KUKA KRL program: MyProgram_023().src

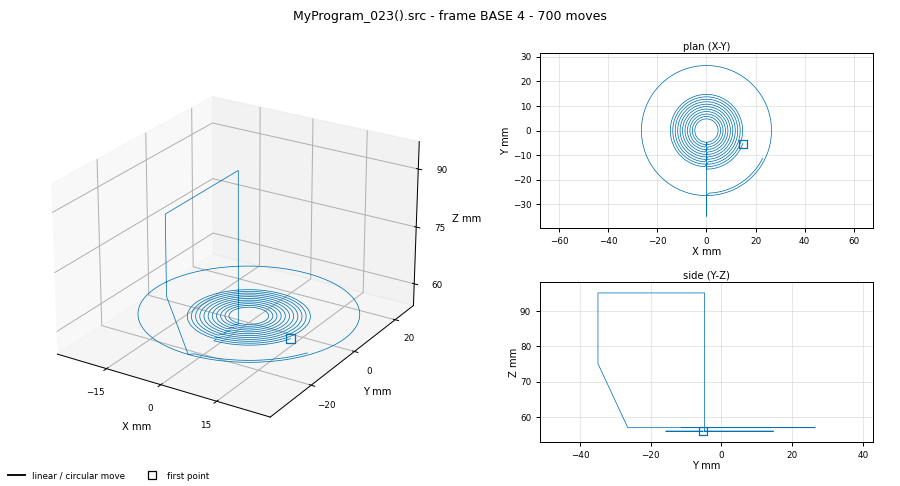
[picture p0: tool path of MyProgram_023().src in frame BASE 4, 700 of 700 moves have a stored position in this frame; points joined in program order, loops and branches not executed]
&ACCESS RVP
&REL 1
&PARAM TEMPLATE = C:\KRC\Roboter\Template\vorgabe
&PARAM EDITMASK = *
DEF MyProgram_023()
; ---- Setting reference (Base) ----
$BASE = BASE_DATA[4]

; --------------------------
; ---- Setting tool (TCP) ----
$TOOL = TOOL_DATA[3]
; --------------------------

$VEL.CP = VEL_APROX_PRINT
Startdeposition()
$VEL.CP = VEL_PRINT
LIN {X 14.8048,Y -5.3302,Z 56,A -29.3112,B 24.8121,C -3.1607,E1 25.1484,E2 -248.3313} C_DIS
LIN {X 13.9602,Y -7.2597,Z 56,A -35.481,B 24.8134,C -3.1503,E1 25.1412,E2 -242.1703} C_DIS
LIN {X 13.4677,Y -8.1371,Z 56,A -39.3253,B 24.8148,C -3.1386,E1 25.1358,E2 -238.3181} C_DIS
LIN {X 12.8219,Y -9.1209,Z 56,A -44.2575,B 24.8167,C -3.122,E1 25.128,E2 -233.371} C_DIS
LIN {X 12.0786,Y -10.0846,Z 56,A -48.5761,B 24.818,C -3.1116,E1 25.1204,E2 -229.0476} C_DIS
LIN {X 11.0622,Y -11.1901,Z 56,A -53.5865,B 24.8191,C -3.1018,E1 25.1107,E2 -224.0359} C_DIS
LIN {X 10.1799,Y -11.9958,Z 56,A -57.8584,B 24.8202,C -3.0927,E1 25.1018,E2 -219.7593} C_DIS
LIN {X 9.2719,Y -12.7131,Z 56,A -62.3619,B 24.8214,C -3.0819,E1 25.0918,E2 -215.2466} C_DIS
LIN {X 8.1629,Y -13.4521,Z 56,A -67.2273,B 24.8225,C -3.0728,E1 25.0803,E2 -210.3752} C_DIS
LIN {X 7.0535,Y -14.0655,Z 56,A -71.7054,B 24.8233,C -3.0661,E1 25.0693,E2 -205.8939} C_DIS
LIN {X 5.5713,Y -14.7154,Z 56,A -78.5194,B 24.8249,C -3.0521,E1 25.0516,E2 -199.062} C_DIS
LIN {X 4.0025,Y -15.2173,Z 56,A -84.3756,B 24.8255,C -3.0465,E1 25.0359,E2 -193.2024} C_DIS
LIN {X 1.9688,Y -15.6113,Z 56,A -91.411,B 24.8258,C -3.044,E1 25.0165,E2 -186.168} C_DIS
LIN {X 0.1829,Y -15.7341,Z 56,A -98.106,B 24.8262,C -3.0407,E1 24.9978,E2 -179.4672} C_DIS
LIN {X 0.1829,Y -15.7341,Z 56,A -98.106,B 24.8262,C -3.0407,E1 24.9978,E2 -179.4672} C_DIS
Enddeposition()
LIN {X 0.0548,Y -14.7363,Z 56,A -95.9481,B 24.8226,C -3.0715,E1 25.004,E2 -181.6985} C_DIS
Startdeposition()
$VEL.CP = VEL_PRINT
LIN {X 1.2094,Y -14.6873,Z 56,A -90.7717,B 24.822,C -3.0772,E1 25.0185,E2 -186.886} C_DIS
LIN {X 3.1948,Y -14.3867,Z 56,A -83.0175,B 24.8213,C -3.083,E1 25.0398,E2 -194.6453} C_DIS
LIN {X 4.7095,Y -13.964,Z 56,A -77.5601,B 24.821,C -3.0859,E1 25.0543,E2 -200.0999} C_DIS
LIN {X 5.781,Y -13.5555,Z 56,A -72.1308,B 24.8195,C -3.0983,E1 25.0684,E2 -205.5461} C_DIS
LIN {X 7.833,Y -12.4829,Z 56,A -64.8508,B 24.8191,C -3.1022,E1 25.0861,E2 -212.8139} C_DIS
LIN {X 8.8701,Y -11.7687,Z 56,A -58.779,B 24.817,C -3.12,E1 25.1,E2 -218.907} C_DIS
LIN {X 9.9895,Y -10.8348,Z 56,A -53.7158,B 24.816,C -3.1283,E1 25.1106,E2 -223.9698} C_DIS
LIN {X 10.8598,Y -9.9602,Z 56,A -49.2201,B 24.8149,C -3.1375,E1 25.1193,E2 -228.4681} C_DIS
LIN {X 11.6373,Y -9.042,Z 56,A -44.418,B 24.8134,C -3.1504,E1 25.1279,E2 -233.2784} C_DIS
LIN {X 12.467,Y -7.8585,Z 56,A -37.7373,B 24.8106,C -3.1737,E1 25.1382,E2 -239.9813} C_DIS
LIN {X 13.1856,Y -6.5817,Z 56,A -32.3096,B 24.8089,C -3.1879,E1 25.1452,E2 -245.4139} C_DIS
LIN {X 13.8526,Y -5.0285,Z 56,A -26.548,B 24.8073,C -3.201,E1 25.1512,E2 -251.1747} C_DIS
LIN {X 14.1872,Y -3.9875,Z 56,A -22.1497,B 24.8056,C -3.2151,E1 25.1547,E2 -255.5813} C_DIS
LIN {X 14.4328,Y -2.9781,Z 56,A -18.2812,B 24.8042,C -3.2262,E1 25.1571,E2 -259.4536} C_DIS
LIN {X 14.6165,Y -1.8806,Z 56,A -13.1649,B 24.8018,C -3.246,E1 25.1591,E2 -264.5866} C_DIS
LIN {X 14.7344,Y -0.2827,Z 56,A -7.0232,B 24.7995,C -3.2646,E1 25.1598,E2 -270.7361} C_DIS
LIN {X 14.6312,Y 1.7639,Z 56,A 0.269,B 24.7972,C -3.2837,E1 25.1582,E2 -278.0303} C_DIS
LIN {X 14.3689,Y 3.2719,Z 56,A 6.2117,B 24.7949,C -3.3016,E1 25.155,E2 -283.9807} C_DIS
LIN {X 13.964,Y 4.709,Z 56,A 12.9283,B 24.7919,C -3.3256,E1 25.1494,E2 -290.716} C_DIS
LIN {X 13.275,Y 6.3989,Z 56,A 18.77,B 24.7907,C -3.3355,E1 25.1428,E2 -296.5494} C_DIS
LIN {X 12.5995,Y 7.6442,Z 56,A 25.1855,B 24.788,C -3.3565,E1 25.1338,E2 -302.9817} C_DIS
LIN {X 11.6707,Y 8.9959,Z 56,A 29.6616,B 24.7878,C -3.3581,E1 25.1266,E2 -307.4397} C_DIS
LIN {X 10.7914,Y 10.0362,Z 56,A 37.2967,B 24.7842,C -3.3862,E1 25.1125,E2 -315.1075} C_DIS
LIN {X 9.6504,Y 11.138,Z 56,A 42.6202,B 24.7834,C -3.3923,E1 25.1014,E2 -320.4241} C_DIS
LIN {X 8.5044,Y 12.0354,Z 56,A 47.752,B 24.7827,C -3.3985,E1 25.09,E2 -325.552} C_DIS
LIN {X 7.3595,Y 12.7674,Z 56,A 53.871,B 24.781,C -3.4113,E1 25.0753,E2 -331.6826} C_DIS
LIN {X 5.1068,Y 13.8238,Z 56,A 64.3115,B 24.7791,C -3.4257,E1 25.0484,E2 -342.133} C_DIS
LIN {X 3.3707,Y 14.3465,Z 56,A 69.8758,B 24.7796,C -3.4218,E1 25.0335,E2 -347.6792} C_DIS
LIN {X 2.2012,Y 14.5718,Z 56,A 74.8904,B 24.7792,C -3.4253,E1 25.0196,E2 -352.6969} C_DIS
LIN {X 0.5459,Y 14.7267,Z 56,A 80.5918,B 24.7796,C -3.4218,E1 25.0038,E2 -358.3873} C_DIS
LIN {X -0.7491,Y 14.7179,Z 56,A 86.5134,B 24.7793,C -3.4244,E1 24.9873,E2 -364.3159} C_DIS
LIN {X -1.8751,Y 14.6172,Z 56,A 90.6939,B 24.7797,C -3.421,E1 24.9757,E2 -368.4912} C_DIS
LIN {X -3.2885,Y 14.3633,Z 56,A 95.6264,B 24.7807,C -3.414,E1 24.9622,E2 -373.4124} C_DIS
LIN {X -4.3601,Y 14.0772,Z 56,A 100.1365,B 24.7811,C -3.4102,E1 24.9501,E2 -377.9208} C_DIS
LIN {X -5.4825,Y 13.6792,Z 56,A 104.5629,B 24.782,C -3.4036,E1 24.9385,E2 -382.3406} C_DIS
LIN {X -6.4904,Y 13.2307,Z 56,A 109.4506,B 24.7826,C -3.3992,E1 24.9262,E2 -387.2301} C_DIS
LIN {X -7.726,Y 12.5494,Z 56,A 115.2787,B 24.7836,C -3.3908,E1 24.9122,E2 -393.0555} C_DIS
LIN {X -9.1952,Y 11.5166,Z 56,A 121.4568,B 24.7857,C -3.3745,E1 24.8983,E2 -399.2167} C_DIS
LIN {X -10.1448,Y 10.6894,Z 56,A 127.0188,B 24.7869,C -3.3654,E1 24.8868,E2 -404.7791} C_DIS
LIN {X -11.2667,Y 9.4995,Z 56,A 133.2509,B 24.7889,C -3.3495,E1 24.8752,E2 -411.0011} C_DIS
LIN {X -12.1246,Y 8.377,Z 56,A 138.6054,B 24.7908,C -3.3348,E1 24.8664,E2 -416.3463} C_DIS
LIN {X -12.8562,Y 7.2042,Z 56,A 144.3048,B 24.7925,C -3.3206,E1 24.8583,E2 -422.0411} C_DIS
LIN {X -13.4172,Y 6.096,Z 56,A 148.769,B 24.7944,C -3.306,E1 24.853,E2 -426.4944} C_DIS
LIN {X -13.8066,Y 5.153,Z 56,A 152.7105,B 24.7959,C -3.2942,E1 24.849,E2 -430.4297} C_DIS
LIN {X -14.0831,Y 4.3412,Z 56,A 156.2898,B 24.7971,C -3.2846,E1 24.8459,E2 -434.0065} C_DIS
LIN {X -14.4046,Y 3.1126,Z 56,A 160.9881,B 24.799,C -3.269,E1 24.8429,E2 -438.6951} C_DIS
LIN {X -14.6238,Y 1.8249,Z 56,A 166.5143,B 24.8008,C -3.2541,E1 24.8406,E2 -444.2183} C_DIS
LIN {X -14.7274,Y 0.4637,Z 56,A 171.4099,B 24.8029,C -3.2369,E1 24.8398,E2 -449.1022} C_DIS
LIN {X -14.7165,Y -0.7763,Z 56,A 176.4141,B 24.8047,C -3.2223,E1 24.8402,E2 -454.1014} C_DIS
LIN {X -14.6103,Y -1.9279,Z 56,A -178.8358,B 24.8063,C -3.209,E1 24.8417,E2 -458.848} C_DIS
LIN {X -14.3442,Y -3.3805,Z 56,A -173.1358,B 24.8084,C -3.1917,E1 24.8449,E2 -464.5403} C_DIS
LIN {X -14.0463,Y -4.4582,Z 56,A -168.0512,B 24.8098,C -3.1805,E1 24.849,E2 -469.6274} C_DIS
LIN {X -13.3291,Y -6.2865,Z 56,A -161.3284,B 24.8125,C -3.1574,E1 24.8563,E2 -476.332} C_DIS
LIN {X -12.9229,Y -7.0841,Z 56,A -156.6672,B 24.8133,C -3.1509,E1 24.8625,E2 -481.0023} C_DIS
LIN {X -11.7295,Y -8.9216,Z 56,A -149.7736,B 24.8162,C -3.1261,E1 24.8733,E2 -487.8708} C_DIS
LIN {X -11.1715,Y -9.6111,Z 56,A -144.1744,B 24.8165,C -3.1243,E1 24.8835,E2 -493.491} C_DIS
LIN {X -9.3084,Y -11.4252,Z 56,A -135.6271,B 24.8193,C -3.1,E1 24.901,E2 -502.0148} C_DIS
LIN {X -8.4511,Y -12.0728,Z 56,A -130.3651,B 24.8197,C -3.0967,E1 24.913,E2 -507.2873} C_DIS
LIN {X -6.7508,Y -13.0998,Z 56,A -123.6353,B 24.8213,C -3.0828,E1 24.9293,E2 -514.0036} C_DIS
LIN {X -5.8273,Y -13.5357,Z 56,A -119.2256,B 24.8216,C -3.0803,E1 24.9405,E2 -518.4179} C_DIS
LIN {X -4.5384,Y -14.0208,Z 56,A -113.6765,B 24.822,C -3.0768,E1 24.9551,E2 -523.9693} C_DIS
LIN {X -2.9742,Y -14.4336,Z 56,A -107.9788,B 24.8227,C -3.071,E1 24.9706,E2 -529.661} C_DIS
LIN {X -1.9619,Y -14.6057,Z 56,A -103.8651,B 24.8227,C -3.0706,E1 24.982,E2 -533.7773} C_DIS
LIN {X -0.703,Y -14.7188,Z 56,A -99.2648,B 24.8229,C -3.069,E1 24.9948,E2 -538.3758} C_DIS
LIN {X -0.703,Y -14.7188,Z 56,A -99.2648,B 24.8229,C -3.069,E1 24.9948,E2 -538.3758} C_DIS
Enddeposition()
LIN {X 0.0882,Y -13.7373,Z 56,A -99.2033,B 24.8225,C -3.0726,E1 24.995,E2 -538.4457} C_DIS
Startdeposition()
$VEL.CP = VEL_PRINT
LIN {X -2.2045,Y -13.5607,Z 56,A -108.546,B 24.8223,C -3.0749,E1 24.9691,E2 -529.1025} C_DIS
LIN {X -3.6611,Y -13.242,Z 56,A -113.9205,B 24.8215,C -3.0814,E1 24.9545,E2 -523.7359} C_DIS
LIN {X -4.8429,Y -12.8549,Z 56,A -118,B 24.8206,C -3.0895,E1 24.9438,E2 -519.6682} C_DIS
LIN {X -5.7969,Y -12.4563,Z 56,A -124.0655,B 24.8207,C -3.0881,E1 24.9282,E2 -513.5848} C_DIS
LIN {X -6.9738,Y -11.8372,Z 56,A -129.4609,B 24.8198,C -3.0959,E1 24.9151,E2 -508.1924} C_DIS
LIN {X -8.2177,Y -11.0106,Z 56,A -135.281,B 24.8185,C -3.107,E1 24.9018,E2 -502.3788} C_DIS
LIN {X -9.1001,Y -10.293,Z 56,A -140.145,B 24.8175,C -3.1154,E1 24.8915,E2 -497.5162} C_DIS
LIN {X -9.9975,Y -9.4238,Z 56,A -145.2366,B 24.8162,C -3.1264,E1 24.8815,E2 -492.4291} C_DIS
LIN {X -10.7189,Y -8.5947,Z 56,A -150.0677,B 24.8151,C -3.1361,E1 24.8728,E2 -487.5991} C_DIS
LIN {X -11.4994,Y -7.5177,Z 56,A -154.969,B 24.8133,C -3.1508,E1 24.865,E2 -482.709} C_DIS
LIN {X -12.258,Y -6.2049,Z 56,A -162.1921,B 24.8115,C -3.1657,E1 24.8553,E2 -475.4836} C_DIS
LIN {X -12.8192,Y -4.9422,Z 56,A -167.9265,B 24.8096,C -3.1818,E1 24.8491,E2 -469.7559} C_DIS
LIN {X -13.2224,Y -3.7266,Z 56,A -171.871,B 24.8075,C -3.1994,E1 24.8458,E2 -465.8309} C_DIS
LIN {X -13.4775,Y -2.6674,Z 56,A -178.6467,B 24.8062,C -3.2099,E1 24.8418,E2 -459.0404} C_DIS
LIN {X -13.6777,Y -1.296,Z 56,A 175.7485,B 24.804,C -3.2278,E1 24.8401,E2 -453.4449} C_DIS
LIN {X -13.7274,Y 0.565,Z 56,A 168.6555,B 24.801,C -3.2527,E1 24.8401,E2 -446.3689} C_DIS
LIN {X -13.6144,Y 1.8474,Z 56,A 163.0023,B 24.799,C -3.269,E1 24.8419,E2 -440.721} C_DIS
LIN {X -13.4072,Y 3.0004,Z 56,A 158.4536,B 24.7971,C -3.2844,E1 24.8444,E2 -436.1826} C_DIS
LIN {X -13.1292,Y 4.048,Z 56,A 153.6733,B 24.7954,C -3.2978,E1 24.8481,E2 -431.4067} C_DIS
LIN {X -12.5255,Y 5.6457,Z 56,A 146.1859,B 24.7928,C -3.3183,E1 24.856,E2 -423.9267} C_DIS
LIN {X -11.7299,Y 7.1534,Z 56,A 139.5054,B 24.7903,C -3.3389,E1 24.8651,E2 -417.2604} C_DIS
LIN {X -11.0348,Y 8.1853,Z 56,A 132.9569,B 24.7888,C -3.3503,E1 24.8758,E2 -410.7074} C_DIS
LIN {X -9.4035,Y 10.0169,Z 56,A 123.6703,B 24.7855,C -3.3764,E1 24.8936,E2 -401.4431} C_DIS
LIN {X -8.4735,Y 10.815,Z 56,A 118.8118,B 24.784,C -3.3877,E1 24.9041,E2 -396.5934} C_DIS
LIN {X -7.5312,Y 11.4909,Z 56,A 113.8264,B 24.7829,C -3.3966,E1 24.9156,E2 -391.6126} C_DIS
LIN {X -6.3763,Y 12.1697,Z 56,A 108.8007,B 24.7815,C -3.4075,E1 24.9278,E2 -386.5983} C_DIS
LIN {X -5.4377,Y 12.617,Z 56,A 103.8915,B 24.7809,C -3.4122,E1 24.9402,E2 -381.6883} C_DIS
LIN {X -4.2833,Y 13.0522,Z 56,A 99.2225,B 24.7799,C -3.42,E1 24.9525,E2 -377.0287} C_DIS
LIN {X -3.3313,Y 13.3291,Z 56,A 94.4774,B 24.7796,C -3.422,E1 24.9653,E2 -372.2812} C_DIS
LIN {X -2.0113,Y 13.5886,Z 56,A 89.4219,B 24.7788,C -3.4282,E1 24.9792,E2 -367.2353} C_DIS
LIN {X -0.6959,Y 13.7213,Z 56,A 83.4729,B 24.7788,C -3.4289,E1 24.9957,E2 -361.2853} C_DIS
LIN {X 0.2866,Y 13.7361,Z 56,A 79.6032,B 24.7785,C -3.4305,E1 25.0065,E2 -357.4199} C_DIS
LIN {X 1.5068,Y 13.6561,Z 56,A 74.0874,B 24.7788,C -3.4283,E1 25.0218,E2 -351.9018} C_DIS
LIN {X 2.9208,Y 13.425,Z 56,A 68.1409,B 24.7791,C -3.4261,E1 25.0381,E2 -345.957} C_DIS
LIN {X 4.6649,Y 12.9228,Z 56,A 59.697,B 24.7804,C -3.4159,E1 25.0606,E2 -337.5044} C_DIS
LIN {X 6.2714,Y 12.2241,Z 56,A 53.4336,B 24.7808,C -3.4132,E1 25.0764,E2 -331.2508} C_DIS
LIN {X 7.31,Y 11.633,Z 56,A 48.2066,B 24.7819,C -3.4046,E1 25.0889,E2 -326.0197} C_DIS
LIN {X 8.7427,Y 10.5986,Z 56,A 42.1869,B 24.7824,C -3.4003,E1 25.1023,E2 -320.0114} C_DIS
LIN {X 9.9736,Y 9.4495,Z 56,A 32.2437,B 24.7866,C -3.3674,E1 25.1221,E2 -310.0319} C_DIS
LIN {X 11.3157,Y 7.7921,Z 56,A 24.0158,B 24.7888,C -3.3506,E1 25.1356,E2 -301.8038} C_DIS
LIN {X 12.4931,Y 5.7173,Z 56,A 15.6873,B 24.7907,C -3.3356,E1 25.1464,E2 -293.4836} C_DIS
LIN {X 12.9049,Y 4.7075,Z 56,A 11.2831,B 24.7921,C -3.3239,E1 25.1509,E2 -289.076} C_DIS
LIN {X 13.2704,Y 3.5574,Z 56,A 6.0217,B 24.7942,C -3.3075,E1 25.1551,E2 -283.8057} C_DIS
LIN {X 13.5032,Y 2.535,Z 56,A 1.2414,B 24.7962,C -3.2913,E1 25.1578,E2 -279.0151} C_DIS
LIN {X 13.6854,Y 1.2119,Z 56,A -3.7214,B 24.7978,C -3.2788,E1 25.1594,E2 -274.0519} C_DIS
LIN {X 13.7354,Y 0.1773,Z 56,A -7.8731,B 24.7993,C -3.2667,E1 25.1598,E2 -269.8962} C_DIS
LIN {X 13.687,Y -1.1935,Z 56,A -14.0401,B 24.8019,C -3.2455,E1 25.1588,E2 -263.7156} C_DIS
LIN {X 13.5157,Y -2.4674,Z 56,A -19.5239,B 24.804,C -3.228,E1 25.1564,E2 -258.2224} C_DIS
LIN {X 13.127,Y -4.0549,Z 56,A -25.7527,B 24.806,C -3.2115,E1 25.1519,E2 -251.9904} C_DIS
LIN {X 12.7794,Y -5.0447,Z 56,A -30.7044,B 24.8081,C -3.1942,E1 25.147,E2 -247.0253} C_DIS
LIN {X 12.2474,Y -6.2256,Z 56,A -35.9164,B 24.8098,C -3.18,E1 25.1407,E2 -241.8075} C_DIS
LIN {X 11.6127,Y -7.3418,Z 56,A -41.0181,B 24.8114,C -3.1669,E1 25.1334,E2 -236.7009} C_DIS
LIN {X 10.9215,Y -8.3359,Z 56,A -45.6641,B 24.8127,C -3.1564,E1 25.1258,E2 -232.0524} C_DIS
LIN {X 10.082,Y -9.3337,Z 56,A -51.3966,B 24.8145,C -3.1408,E1 25.1152,E2 -226.3088} C_DIS
LIN {X 9.1447,Y -10.2537,Z 56,A -57.3574,B 24.8164,C -3.125,E1 25.1031,E2 -220.335} C_DIS
LIN {X 8.074,Y -11.116,Z 56,A -62.3643,B 24.8172,C -3.1179,E1 25.092,E2 -215.3294} C_DIS
LIN {X 7.3076,Y -11.6345,Z 56,A -67.32,B 24.8189,C -3.1038,E1 25.0803,E2 -210.3564} C_DIS
LIN {X 5.4767,Y -12.5999,Z 56,A -75.3509,B 24.82,C -3.0939,E1 25.0601,E2 -202.3232} C_DIS
LIN {X 3.8332,Y -13.1933,Z 56,A -82.8593,B 24.8212,C -3.084,E1 25.0402,E2 -194.8057} C_DIS
LIN {X 2.3245,Y -13.5406,Z 56,A -88.9914,B 24.8216,C -3.0803,E1 25.0234,E2 -188.6722} C_DIS
LIN {X 1.0278,Y -13.7006,Z 56,A -94.9502,B 24.8222,C -3.075,E1 25.0068,E2 -182.7043} C_DIS
LIN {X 0.0882,Y -13.7373,Z 56,A -99.2033,B 24.8225,C -3.0726,E1 24.995,E2 -178.4457} C_DIS
Enddeposition()
LIN {X 0.0882,Y -13.7373,Z 56,A -99.2033,B 24.8225,C -3.0726,E1 24.995,E2 -178.4457} C_DIS
Startdeposition()
$VEL.CP = VEL_PRINT
LIN {X 0.846,Y -12.7129,Z 56,A -92.2496,B 24.8185,C -3.1072,E1 25.0146,E2 -185.4806} C_DIS
LIN {X 2.1074,Y -12.5656,Z 56,A -85.9473,B 24.8177,C -3.114,E1 25.032,E2 -191.7932} C_DIS
LIN {X 3.68,Y -12.1981,Z 56,A -79.2495,B 24.8172,C -3.1184,E1 25.0501,E2 -198.491} C_DIS
LIN {X 4.7745,Y -11.8127,Z 56,A -73.2317,B 24.8158,C -3.1298,E1 25.0658,E2 -204.5228} C_DIS
LIN {X 6.5926,Y -10.903,Z 56,A -65.1697,B 24.8148,C -3.1386,E1 25.0856,E2 -212.5827} C_DIS
LIN {X 7.6738,Y -10.171,Z 56,A -58.5287,B 24.8128,C -3.1551,E1 25.1007,E2 -219.2397} C_DIS
LIN {X 8.7439,Y -9.2671,Z 56,A -51.5317,B 24.8106,C -3.174,E1 25.1151,E2 -226.2531} C_DIS
LIN {X 10.2047,Y -7.6288,Z 56,A -42.9898,B 24.8086,C -3.1898,E1 25.1303,E2 -234.7934} C_DIS
LIN {X 10.9664,Y -6.4864,Z 56,A -36.3429,B 24.8062,C -3.2101,E1 25.1402,E2 -241.4548} C_DIS
LIN {X 11.5007,Y -5.4837,Z 56,A -31.1854,B 24.8044,C -3.2252,E1 25.1466,E2 -246.6204} C_DIS
LIN {X 12.1365,Y -3.8775,Z 56,A -25.0553,B 24.803,C -3.2366,E1 25.1525,E2 -252.7433} C_DIS
LIN {X 12.3867,Y -2.9845,Z 56,A -20.1005,B 24.8007,C -3.255,E1 25.1561,E2 -257.7132} C_DIS
LIN {X 12.5465,Y -2.2183,Z 56,A -16.2178,B 24.799,C -3.2686,E1 25.158,E2 -261.6055} C_DIS
LIN {X 12.7239,Y -0.6578,Z 56,A -9.0136,B 24.7962,C -3.2916,E1 25.1597,E2 -268.8215} C_DIS
LIN {X 12.7133,Y 0.84,Z 56,A -2.7132,B 24.794,C -3.3092,E1 25.1591,E2 -275.1263} C_DIS
LIN {X 12.5589,Y 2.1475,Z 56,A 4.0308,B 24.791,C -3.3332,E1 25.1563,E2 -281.8875} C_DIS
LIN {X 12.0597,Y 4.1104,Z 56,A 11.3207,B 24.7892,C -3.3469,E1 25.1509,E2 -289.168} C_DIS
LIN {X 11.6949,Y 5.0558,Z 56,A 16.5606,B 24.787,C -3.3645,E1 25.1454,E2 -294.4206} C_DIS
LIN {X 11.0719,Y 6.3047,Z 56,A 23.0344,B 24.7847,C -3.3824,E1 25.1369,E2 -300.9029} C_DIS
LIN {X 10.4017,Y 7.3581,Z 56,A 28.2429,B 24.7833,C -3.3936,E1 25.1289,E2 -306.1121} C_DIS
LIN {X 9.8575,Y 8.0724,Z 56,A 33.2066,B 24.7813,C -3.4089,E1 25.1202,E2 -311.0889} C_DIS
LIN {X 8.6383,Y 9.3654,Z 56,A 40.2128,B 24.78,C -3.4191,E1 25.1064,E2 -318.0897} C_DIS
LIN {X 7.5062,Y 10.2953,Z 56,A 47.3336,B 24.7781,C -3.4339,E1 25.0907,E2 -325.2192} C_DIS
LIN {X 6.5786,Y 10.9114,Z 56,A 52.0428,B 24.7773,C -3.4396,E1 25.0796,E2 -329.927} C_DIS
LIN {X 5.4854,Y 11.4997,Z 56,A 57.6724,B 24.7764,C -3.4467,E1 25.0656,E2 -335.5582} C_DIS
LIN {X 4.2005,Y 12.0286,Z 56,A 64.408,B 24.7753,C -3.455,E1 25.048,E2 -342.2989} C_DIS
LIN {X 2.9819,Y 12.3873,Z 56,A 69.945,B 24.775,C -3.4575,E1 25.033,E2 -347.8334} C_DIS
LIN {X 1.5044,Y 12.652,Z 56,A 76.7474,B 24.7747,C -3.4595,E1 25.0143,E2 -354.6343} C_DIS
LIN {X 0.0834,Y 12.7408,Z 56,A 82.7812,B 24.775,C -3.4575,E1 24.9974,E2 -360.6618} C_DIS
LIN {X -1.2068,Y 12.6837,Z 56,A 88.7478,B 24.7752,C -3.4557,E1 24.9808,E2 -366.6264} C_DIS
LIN {X -2.5336,Y 12.4865,Z 56,A 94.8571,B 24.7758,C -3.4516,E1 24.9641,E2 -372.732} C_DIS
LIN {X -3.5731,Y 12.2296,Z 56,A 99.4798,B 24.7765,C -3.4461,E1 24.9516,E2 -377.3488} C_DIS
LIN {X -4.7424,Y 11.8255,Z 56,A 105.282,B 24.7773,C -3.4398,E1 24.9365,E2 -383.1479} C_DIS
LIN {X -5.5626,Y 11.4627,Z 56,A 110.2068,B 24.7778,C -3.436,E1 24.9241,E2 -388.0764} C_DIS
LIN {X -7.3339,Y 10.4187,Z 56,A 118.1935,B 24.7804,C -3.4161,E1 24.9053,E2 -396.041} C_DIS
LIN {X -8.226,Y 9.7299,Z 56,A 123.5553,B 24.7817,C -3.4061,E1 24.8937,E2 -401.3989} C_DIS
LIN {X -9.1126,Y 8.9049,Z 56,A 128.9947,B 24.7833,C -3.3935,E1 24.8829,E2 -406.831} C_DIS
LIN {X -9.9217,Y 7.9936,Z 56,A 134.7244,B 24.785,C -3.3803,E1 24.8726,E2 -412.5552} C_DIS
LIN {X -10.7926,Y 6.7713,Z 56,A 141.1342,B 24.7874,C -3.3617,E1 24.8626,E2 -418.9523} C_DIS
LIN {X -11.431,Y 5.627,Z 56,A 147.1457,B 24.7895,C -3.3451,E1 24.8547,E2 -424.9561} C_DIS
LIN {X -11.8217,Y 4.7523,Z 56,A 151.5735,B 24.791,C -3.3326,E1 24.85,E2 -429.3785} C_DIS
LIN {X -12.2361,Y 3.551,Z 56,A 156.9921,B 24.7932,C -3.3151,E1 24.8453,E2 -434.786} C_DIS
LIN {X -12.5152,Y 2.3885,Z 56,A 162.5489,B 24.7953,C -3.2988,E1 24.842,E2 -440.3364} C_DIS
LIN {X -12.6745,Y 1.3008,Z 56,A 168.055,B 24.7971,C -3.2841,E1 24.8402,E2 -445.8401} C_DIS
LIN {X -12.7392,Y -0.2228,Z 56,A 174.5894,B 24.7998,C -3.2624,E1 24.8399,E2 -452.362} C_DIS
LIN {X -12.6656,Y -1.3839,Z 56,A 179.7288,B 24.8018,C -3.2462,E1 24.8411,E2 -457.4934} C_DIS
LIN {X -12.5123,Y -2.4001,Z 56,A -175.4287,B 24.8035,C -3.2326,E1 24.8434,E2 -462.3319} C_DIS
LIN {X -12.1912,Y -3.7032,Z 56,A -170.2033,B 24.8058,C -3.2138,E1 24.8472,E2 -467.5427} C_DIS
LIN {X -11.8078,Y -4.7856,Z 56,A -164.107,B 24.8074,C -3.2004,E1 24.8531,E2 -473.6413} C_DIS
LIN {X -11.2481,Y -5.984,Z 56,A -158.033,B 24.8093,C -3.1847,E1 24.8607,E2 -479.7103} C_DIS
LIN {X -10.3963,Y -7.3652,Z 56,A -150.7404,B 24.8114,C -3.1666,E1 24.8718,E2 -486.9962} C_DIS
LIN {X -9.5188,Y -8.4686,Z 56,A -143.7134,B 24.813,C -3.1539,E1 24.8845,E2 -494.0249} C_DIS
LIN {X -8.0975,Y -9.8364,Z 56,A -135.2277,B 24.8151,C -3.136,E1 24.9021,E2 -502.5018} C_DIS
LIN {X -6.9871,Y -10.6542,Z 56,A -129.0524,B 24.8163,C -3.1261,E1 24.9162,E2 -508.6743} C_DIS
LIN {X -6.1846,Y -11.1395,Z 56,A -125.0349,B 24.817,C -3.1199,E1 24.926,E2 -512.6888} C_DIS
LIN {X -5.3265,Y -11.5744,Z 56,A -120.8363,B 24.8176,C -3.1145,E1 24.9366,E2 -516.8854} C_DIS
LIN {X -4.0768,Y -12.0712,Z 56,A -114.3431,B 24.8181,C -3.1109,E1 24.9536,E2 -523.383} C_DIS
LIN {X -2.7873,Y -12.4323,Z 56,A -108.7352,B 24.8186,C -3.1061,E1 24.9687,E2 -528.9875} C_DIS
LIN {X -1.7393,Y -12.6219,Z 56,A -104.0183,B 24.8188,C -3.1045,E1 24.9818,E2 -533.7049} C_DIS
LIN {X -0.655,Y -12.7241,Z 56,A -98.9908,B 24.8188,C -3.1051,E1 24.9958,E2 -538.7358} C_DIS
LIN {X -0.655,Y -12.7241,Z 56,A -98.9908,B 24.8188,C -3.1051,E1 24.9958,E2 -538.7358} C_DIS
Enddeposition()
LIN {X 0.0689,Y -11.7371,Z 56,A -96.9233,B 24.8172,C -3.1177,E1 25.0016,E2 -540.8333} C_DIS
Startdeposition()
$VEL.CP = VEL_PRINT
LIN {X -0.9726,Y -11.7024,Z 56,A -103.1695,B 24.8178,C -3.1127,E1 24.9842,E2 -534.5737} C_DIS
LIN {X -2.0877,Y -11.556,Z 56,A -109.1817,B 24.8178,C -3.1122,E1 24.9676,E2 -528.5551} C_DIS
LIN {X -3.0518,Y -11.3394,Z 56,A -114.07,B 24.8176,C -3.1146,E1 24.9543,E2 -523.6655} C_DIS
LIN {X -4.533,Y -10.8325,Z 56,A -121.9664,B 24.8169,C -3.1206,E1 24.9337,E2 -515.7672} C_DIS
LIN {X -5.6889,Y -10.2731,Z 56,A -127.7671,B 24.8159,C -3.1295,E1 24.9193,E2 -509.9718} C_DIS
LIN {X -6.6994,Y -9.6409,Z 56,A -133.2843,B 24.8147,C -3.139,E1 24.9065,E2 -504.4593} C_DIS
LIN {X -7.3672,Y -9.1412,Z 56,A -137.3038,B 24.8139,C -3.1461,E1 24.8976,E2 -500.4421} C_DIS
LIN {X -7.9978,Y -8.5953,Z 56,A -141.4431,B 24.813,C -3.1538,E1 24.889,E2 -496.3045} C_DIS
LIN {X -8.5875,Y -8.0055,Z 56,A -145.4987,B 24.812,C -3.1622,E1 24.8811,E2 -492.2518} C_DIS
LIN {X -9.1346,Y -7.376,Z 56,A -149.6163,B 24.8109,C -3.1713,E1 24.8737,E2 -488.1368} C_DIS
LIN {X -9.7547,Y -6.5378,Z 56,A -154.9489,B 24.8095,C -3.1831,E1 24.8652,E2 -482.8066} C_DIS
LIN {X -10.2644,Y -5.7047,Z 56,A -160.3975,B 24.8081,C -3.1947,E1 24.8576,E2 -477.3572} C_DIS
LIN {X -10.9919,Y -4.1321,Z 56,A -167.9347,B 24.8051,C -3.2189,E1 24.8492,E2 -469.8364} C_DIS
LIN {X -11.5022,Y -2.3647,Z 56,A -178.9176,B 24.8021,C -3.2439,E1 24.8417,E2 -458.8496} C_DIS
LIN {X -11.7262,Y -0.6128,Z 56,A 173.2612,B 24.7988,C -3.2709,E1 24.8398,E2 -451.046} C_DIS
LIN {X -11.6918,Y 1.0956,Z 56,A 164.8812,B 24.7955,C -3.2967,E1 24.8411,E2 -442.6777} C_DIS
LIN {X -11.4868,Y 2.4409,Z 56,A 158.8117,B 24.7929,C -3.3175,E1 24.8441,E2 -436.6221} C_DIS
LIN {X -11.2026,Y 3.5215,Z 56,A 153.0503,B 24.7909,C -3.3339,E1 24.8486,E2 -430.8665} C_DIS
LIN {X -10.7955,Y 4.6202,Z 56,A 147.3153,B 24.7888,C -3.3507,E1 24.8545,E2 -425.14} C_DIS
LIN {X -10.2689,Y 5.6967,Z 56,A 142.136,B 24.7866,C -3.3679,E1 24.8611,E2 -419.9742} C_DIS
LIN {X -9.5216,Y 6.8732,Z 56,A 133.2496,B 24.7845,C -3.384,E1 24.8751,E2 -411.0824} C_DIS
LIN {X -7.9763,Y 8.6186,Z 56,A 122.0094,B 24.781,C -3.411,E1 24.8969,E2 -399.8587} C_DIS
LIN {X -6.8958,Y 9.5049,Z 56,A 115.5157,B 24.7792,C -3.4253,E1 24.9114,E2 -393.3759} C_DIS
LIN {X -5.2981,Y 10.4799,Z 56,A 107.467,B 24.7769,C -3.4429,E1 24.9309,E2 -385.3458} C_DIS
LIN {X -4.3393,Y 10.9121,Z 56,A 101.5841,B 24.7762,C -3.4482,E1 24.946,E2 -379.4621} C_DIS
LIN {X -2.8904,Y 11.3818,Z 56,A 94.6219,B 24.775,C -3.4573,E1 24.9647,E2 -372.5101} C_DIS
LIN {X -1.571,Y 11.6375,Z 56,A 87.6205,B 24.7746,C -3.4605,E1 24.9839,E2 -365.5099} C_DIS
LIN {X -0.3179,Y 11.7389,Z 56,A 81.9891,B 24.7741,C -3.4644,E1 24.9996,E2 -359.8861} C_DIS
LIN {X 0.7997,Y 11.7158,Z 56,A 76.2345,B 24.7742,C -3.4635,E1 25.0157,E2 -354.1314} C_DIS
LIN {X 2.0147,Y 11.5691,Z 56,A 70.2249,B 24.7744,C -3.4618,E1 25.0322,E2 -348.1231} C_DIS
LIN {X 3.2337,Y 11.289,Z 56,A 64.5724,B 24.7746,C -3.4602,E1 25.0475,E2 -342.4753} C_DIS
LIN {X 4.1701,Y 10.9771,Z 56,A 59.0303,B 24.7756,C -3.4526,E1 25.0621,E2 -336.9268} C_DIS
LIN {X 5.8427,Y 10.1864,Z 56,A 50.4083,B 24.7768,C -3.4435,E1 25.0835,E2 -328.3067} C_DIS
LIN {X 6.9689,Y 9.4518,Z 56,A 44.2671,B 24.7779,C -3.4352,E1 25.0976,E2 -322.1668} C_DIS
LIN {X 7.932,Y 8.6594,Z 56,A 37.6415,B 24.7798,C -3.4208,E1 25.1116,E2 -315.5329} C_DIS
LIN {X 8.7174,Y 7.8682,Z 56,A 32.1301,B 24.7813,C -3.4088,E1 25.1221,E2 -310.017} C_DIS
LIN {X 9.7238,Y 6.584,Z 56,A 24.1917,B 24.7837,C -3.3899,E1 25.1352,E2 -302.0722} C_DIS
LIN {X 10.515,Y 5.2281,Z 56,A 16.7782,B 24.7861,C -3.3714,E1 25.1451,E2 -294.6534} C_DIS
LIN {X 11.0579,Y 3.9525,Z 56,A 10.0932,B 24.7885,C -3.3529,E1 25.1519,E2 -287.9616} C_DIS
LIN {X 11.3944,Y 2.8409,Z 56,A 4.7855,B 24.7903,C -3.3386,E1 25.1559,E2 -282.6506} C_DIS
LIN {X 11.593,Y 1.8704,Z 56,A -0.1487,B 24.7922,C -3.3234,E1 25.1583,E2 -277.7091} C_DIS
LIN {X 11.7215,Y 0.706,Z 56,A -5.447,B 24.7941,C -3.3086,E1 25.1596,E2 -272.4072} C_DIS
LIN {X 11.7141,Y -0.8229,Z 56,A -13.0618,B 24.7971,C -3.2844,E1 25.1591,E2 -264.7803} C_DIS
LIN {X 11.5493,Y -2.1251,Z 56,A -19.7989,B 24.7998,C -3.2623,E1 25.1563,E2 -258.0303} C_DIS
LIN {X 11.2431,Y -3.3904,Z 56,A -25.3163,B 24.8015,C -3.2485,E1 25.1523,E2 -252.5121} C_DIS
LIN {X 10.9547,Y -4.2298,Z 56,A -30.1052,B 24.8035,C -3.2325,E1 25.1478,E2 -247.7119} C_DIS
LIN {X 10.4428,Y -5.3654,Z 56,A -34.8196,B 24.8045,C -3.224,E1 25.1422,E2 -243.0029} C_DIS
LIN {X 9.9467,Y -6.242,Z 56,A -41.6782,B 24.8077,C -3.1975,E1 25.1325,E2 -236.1166} C_DIS
LIN {X 9.1352,Y -7.3789,Z 56,A -48.1538,B 24.8096,C -3.1819,E1 25.1215,E2 -229.6348} C_DIS
LIN {X 8.2431,Y -8.3638,Z 56,A -54.2695,B 24.8112,C -3.1686,E1 25.1097,E2 -223.514} C_DIS
LIN {X 7.4207,Y -9.1011,Z 56,A -59.6999,B 24.8126,C -3.1565,E1 25.0982,E2 -218.0762} C_DIS
LIN {X 6.4532,Y -9.8111,Z 56,A -64.9778,B 24.8136,C -3.1483,E1 25.0861,E2 -212.797} C_DIS
LIN {X 5.2093,Y -10.5243,Z 56,A -72.7678,B 24.8155,C -3.1322,E1 25.067,E2 -204.9912} C_DIS
LIN {X 4.0383,Y -11.0268,Z 56,A -78.8324,B 24.8164,C -3.1246,E1 25.0512,E2 -198.922} C_DIS
LIN {X 2.6585,Y -11.4381,Z 56,A -86.2807,B 24.8175,C -3.1154,E1 25.0311,E2 -191.4637} C_DIS
LIN {X 0.9818,Y -11.7016,Z 56,A -93.8354,B 24.8177,C -3.1135,E1 25.0102,E2 -183.9103} C_DIS
LIN {X 0.0689,Y -11.7371,Z 56,A -96.9233,B 24.8172,C -3.1177,E1 25.0016,E2 -180.8333} C_DIS
Enddeposition()
LIN {X 0.0689,Y -11.7371,Z 56,A -96.9233,B 24.8172,C -3.1177,E1 25.0016,E2 -180.8333} C_DIS
Startdeposition()
$VEL.CP = VEL_PRINT
LIN {X 0.4819,Y -10.7343,Z 56,A -92.7327,B 24.8142,C -3.1434,E1 25.0135,E2 -185.0837} C_DIS
LIN {X 2.1779,Y -10.5217,Z 56,A -84.8318,B 24.8141,C -3.1445,E1 25.0353,E2 -192.9798} C_DIS
LIN {X 3.5686,Y -10.1349,Z 56,A -75.7142,B 24.8122,C -3.1599,E1 25.0596,E2 -202.1177} C_DIS
LIN {X 5.1038,Y -9.4556,Z 56,A -67.7535,B 24.8112,C -3.1687,E1 25.0796,E2 -210.0783} C_DIS
LIN {X 6.0628,Y -8.8714,Z 56,A -62.4013,B 24.8103,C -3.1763,E1 25.0922,E2 -215.4315} C_DIS
LIN {X 7.2221,Y -7.9562,Z 56,A -52.4324,B 24.8067,C -3.2056,E1 25.1135,E2 -225.4312} C_DIS
LIN {X 8.4512,Y -6.6355,Z 56,A -44.354,B 24.805,C -3.2201,E1 25.1282,E2 -233.5075} C_DIS
LIN {X 9.1708,Y -5.594,Z 56,A -39.0508,B 24.8039,C -3.2293,E1 25.1365,E2 -238.8063} C_DIS
LIN {X 9.6542,Y -4.7172,Z 56,A -31.5702,B 24.8003,C -3.2582,E1 25.1462,E2 -246.316} C_DIS
LIN {X 10.2192,Y -3.3118,Z 56,A -25.7546,B 24.7992,C -3.2675,E1 25.152,E2 -252.1213} C_DIS
LIN {X 10.4244,Y -2.6067,Z 56,A -20.1964,B 24.7963,C -3.2903,E1 25.1561,E2 -257.7014} C_DIS
LIN {X 10.6471,Y -1.4317,Z 56,A -14.4932,B 24.7944,C -3.3056,E1 25.1587,E2 -263.4075} C_DIS
LIN {X 10.7433,Y -0.1964,Z 56,A -7.2552,B 24.7913,C -3.3303,E1 25.1598,E2 -270.6611} C_DIS
LIN {X 10.6861,Y 1.124,Z 56,A -0.2014,B 24.7886,C -3.352,E1 25.1583,E2 -277.7246} C_DIS
LIN {X 10.4459,Y 2.5184,Z 56,A 8.3722,B 24.7849,C -3.3813,E1 25.1533,E2 -286.3179} C_DIS
LIN {X 9.8259,Y 4.3484,Z 56,A 17.0712,B 24.7824,C -3.4001,E1 25.1447,E2 -295.013} C_DIS
LIN {X 9.3125,Y 5.3554,Z 56,A 22.9977,B 24.7805,C -3.4154,E1 25.1369,E2 -300.9448} C_DIS
LIN {X 8.6214,Y 6.4133,Z 56,A 30.1632,B 24.778,C -3.4343,E1 25.1255,E2 -308.12} C_DIS
LIN {X 7.8893,Y 7.2951,Z 56,A 36.0264,B 24.7765,C -3.4463,E1 25.1147,E2 -313.9853} C_DIS
LIN {X 7.1278,Y 8.0406,Z 56,A 41.8666,B 24.7749,C -3.4584,E1 25.1027,E2 -319.8303} C_DIS
LIN {X 6.4485,Y 8.595,Z 56,A 46.6506,B 24.7737,C -3.467,E1 25.0921,E2 -324.6175} C_DIS
LIN {X 5.3919,Y 9.2943,Z 56,A 52.5305,B 24.773,C -3.4727,E1 25.0782,E2 -330.4919} C_DIS
LIN {X 4.5822,Y 9.7192,Z 56,A 58.1442,B 24.7718,C -3.482,E1 25.0642,E2 -336.1128} C_DIS
LIN {X 3.7406,Y 10.0729,Z 56,A 62.8258,B 24.7713,C -3.4858,E1 25.052,E2 -340.793} C_DIS
LIN {X 2.6366,Y 10.4166,Z 56,A 68.7806,B 24.7709,C -3.489,E1 25.036,E2 -346.7455} C_DIS
LIN {X 1.3708,Y 10.6571,Z 56,A 75.8729,B 24.7705,C -3.492,E1 25.0165,E2 -353.8379} C_DIS
LIN {X 0.2673,Y 10.7419,Z 56,A 81.9512,B 24.7705,C -3.4923,E1 24.9995,E2 -359.915} C_DIS
LIN {X -1.1404,Y 10.6843,Z 56,A 90.4418,B 24.7705,C -3.4921,E1 24.9759,E2 -368.4087} C_DIS
LIN {X -2.9142,Y 10.3422,Z 56,A 98.2825,B 24.7722,C -3.479,E1 24.9546,E2 -376.2281} C_DIS
LIN {X -3.7947,Y 10.0525,Z 56,A 103.2682,B 24.7729,C -3.4732,E1 24.9415,E2 -381.2095} C_DIS
LIN {X -4.5887,Y 9.7162,Z 56,A 108.6139,B 24.7736,C -3.4681,E1 24.9279,E2 -386.5559} C_DIS
LIN {X -5.4498,Y 9.2604,Z 56,A 114.7906,B 24.7745,C -3.461,E1 24.9129,E2 -392.734} C_DIS
LIN {X -6.94,Y 8.2032,Z 56,A 123.1892,B 24.7774,C -3.4392,E1 24.8943,E2 -401.1107} C_DIS
LIN {X -7.6987,Y 7.4916,Z 56,A 128.6713,B 24.779,C -3.4265,E1 24.8833,E2 -406.585} C_DIS
LIN {X -8.6053,Y 6.4349,Z 56,A 137.1307,B 24.7813,C -3.4086,E1 24.8685,E2 -415.0411} C_DIS
LIN {X -9.2855,Y 5.4074,Z 56,A 143.1078,B 24.7837,C -3.3902,E1 24.8597,E2 -421.0045} C_DIS
LIN {X -9.7659,Y 4.4819,Z 56,A 148.8633,B 24.7857,C -3.3743,E1 24.8527,E2 -426.7532} C_DIS
LIN {X -10.0943,Y 3.6824,Z 56,A 153.4686,B 24.7875,C -3.3607,E1 24.8481,E2 -431.3516} C_DIS
LIN {X -10.4089,Y 2.6669,Z 56,A 159.413,B 24.7897,C -3.3436,E1 24.8437,E2 -437.2895} C_DIS
LIN {X -10.6356,Y 1.5308,Z 56,A 165.1557,B 24.7921,C -3.3243,E1 24.841,E2 -443.02} C_DIS
LIN {X -10.7385,Y 0.3747,Z 56,A 171.5766,B 24.7945,C -3.3052,E1 24.8398,E2 -449.4337} C_DIS
LIN {X -10.7099,Y -0.8692,Z 56,A 178.538,B 24.797,C -3.2849,E1 24.8408,E2 -456.3882} C_DIS
LIN {X -10.5772,Y -1.8903,Z 56,A -175.8413,B 24.7991,C -3.2684,E1 24.8433,E2 -462.0027} C_DIS
LIN {X -10.2439,Y -3.2428,Z 56,A -168.3565,B 24.8017,C -3.2466,E1 24.8489,E2 -469.4788} C_DIS
LIN {X -9.7539,Y -4.5077,Z 56,A -161.4474,B 24.8042,C -3.2263,E1 24.8563,E2 -476.3775} C_DIS
LIN {X -9.3284,Y -5.3328,Z 56,A -155.9874,B 24.8057,C -3.2139,E1 24.8637,E2 -481.8364} C_DIS
LIN {X -8.6633,Y -6.3565,Z 56,A -150.6348,B 24.8078,C -3.1967,E1 24.8721,E2 -487.1745} C_DIS
LIN {X -7.9065,Y -7.2756,Z 56,A -143.1008,B 24.8093,C -3.1843,E1 24.8858,E2 -494.713} C_DIS
LIN {X -6.8664,Y -8.2643,Z 56,A -134.7494,B 24.8109,C -3.1711,E1 24.9033,E2 -503.0657} C_DIS
LIN {X -5.5564,Y -9.1967,Z 56,A -126.926,B 24.8126,C -3.1565,E1 24.9215,E2 -510.8799} C_DIS
LIN {X -4.4812,Y -9.766,Z 56,A -120.5522,B 24.8136,C -3.1486,E1 24.9375,E2 -517.2515} C_DIS
LIN {X -3.3531,Y -10.2084,Z 56,A -114.6636,B 24.8144,C -3.1415,E1 24.9529,E2 -523.1352} C_DIS
LIN {X -2.1245,Y -10.5329,Z 56,A -107.4587,B 24.8147,C -3.1394,E1 24.9725,E2 -530.3448} C_DIS
LIN {X -1.1499,Y -10.6832,Z 56,A -102.1048,B 24.8147,C -3.1388,E1 24.9873,E2 -535.7012} C_DIS
LIN {X 0.0476,Y -10.7445,Z 56,A -98.8074,B 24.816,C -3.1282,E1 24.9964,E2 -538.9743} C_DIS
Enddeposition()
LIN {X 0.0339,Y -9.7462,Z 56,A -3.055,B 0,C 0,E1 0.1598,E2 -629.9288} C_DIS
Startdeposition()
$VEL.CP = VEL_PRINT
LIN {X -1.0348,Y -9.6918,Z 56,A -3.092,B 0,C 0,E1 0.1598,E2 -629.9286} C_DIS
LIN {X -2.5534,Y -9.4064,Z 56,A -3.1354,B 0,C 0,E1 0.1598,E2 -629.9286} C_DIS
LIN {X -3.7158,Y -9.011,Z 56,A -3.1611,B 0,C 0,E1 0.1598,E2 -629.9287} C_DIS
LIN {X -4.6425,Y -8.5697,Z 56,A -3.1763,B 0,C 0,E1 0.1598,E2 -629.9287} C_DIS
LIN {X -5.7951,Y -7.8372,Z 56,A -3.1872,B 0,C 0,E1 0.1598,E2 -629.929} C_DIS
LIN {X -6.704,Y -7.0756,Z 56,A -3.1881,B 0,C 0,E1 0.1598,E2 -629.929} C_DIS
LIN {X -7.541,Y -6.1758,Z 56,A -3.1804,B 0,C 0,E1 0.1598,E2 -629.9291} C_DIS
LIN {X -8.0538,Y -5.4904,Z 56,A -3.1703,B 0,C 0,E1 0.1598,E2 -629.9289} C_DIS
LIN {X -8.6702,Y -4.4467,Z 56,A -3.1483,B 0,C 0,E1 0.1598,E2 -629.9293} C_DIS
LIN {X -9.0134,Y -3.7099,Z 56,A -3.1298,B 0,C 0,E1 0.1598,E2 -629.929} C_DIS
LIN {X -9.4353,Y -2.4451,Z 56,A -3.0914,B 0,C 0,E1 0.1598,E2 -629.9293} C_DIS
LIN {X -9.6328,Y -1.4612,Z 56,A -3.0572,B 0,C 0,E1 0.1598,E2 -629.929} C_DIS
LIN {X -9.7423,Y -0.3063,Z 56,A -3.0121,B 0,C 0,E1 0.1598,E2 -629.9291} C_DIS
LIN {X -9.7093,Y 0.8574,Z 56,A -2.9616,B 0,C 0,E1 0.1598,E2 -629.9291} C_DIS
LIN {X -9.5398,Y 2.0003,Z 56,A -2.907,B 0,C 0,E1 0.1598,E2 -629.929} C_DIS
LIN {X -9.2331,Y 3.1236,Z 56,A -2.848,B 0,C 0,E1 0.1598,E2 -629.929} C_DIS
LIN {X -8.7816,Y 4.2294,Z 56,A -2.7848,B 0,C 0,E1 0.1598,E2 -629.9287} C_DIS
LIN {X -7.9512,Y 5.6372,Z 56,A -2.6942,B 0,C 0,E1 0.1598,E2 -629.929} C_DIS
LIN {X -7.0946,Y 6.6839,Z 56,A -2.6187,B 0,C 0,E1 0.1598,E2 -629.9285} C_DIS
LIN {X -6.3552,Y 7.3904,Z 56,A -2.5618,B 0,C 0,E1 0.1598,E2 -629.9281} C_DIS
LIN {X -4.9254,Y 8.4111,Z 56,A -2.4655,B 0,C 0,E1 0.1598,E2 -629.9282} C_DIS
LIN {X -3.7907,Y 8.9798,Z 56,A -2.3998,B 0,C 0,E1 0.1598,E2 -629.9278} C_DIS
LIN {X -2.711,Y 9.3593,Z 56,A -2.344,B 0,C 0,E1 0.1598,E2 -629.9276} C_DIS
LIN {X -1.9178,Y 9.5518,Z 56,A -2.3066,B 0,C 0,E1 0.1598,E2 -629.9276} C_DIS
LIN {X -0.9091,Y 9.7046,Z 56,A -2.2628,B 0,C 0,E1 0.1598,E2 -629.9275} C_DIS
LIN {X 0.438,Y 9.7369,Z 56,A -2.2117,B 0,C 0,E1 0.1598,E2 -629.9274} C_DIS
LIN {X 1.7552,Y 9.5877,Z 56,A -2.1693,B 0,C 0,E1 0.1598,E2 -629.9274} C_DIS
LIN {X 2.7081,Y 9.3633,Z 56,A -2.1437,B 0,C 0,E1 0.1598,E2 -629.9274} C_DIS
LIN {X 3.4311,Y 9.1231,Z 56,A -2.1272,B 0,C 0,E1 0.1598,E2 -629.9274} C_DIS
LIN {X 4.4692,Y 8.6621,Z 56,A -2.1084,B 0,C 0,E1 0.1598,E2 -629.9274} C_DIS
LIN {X 5.2418,Y 8.2177,Z 56,A -2.0988,B 0,C 0,E1 0.1598,E2 -629.9274} C_DIS
LIN {X 6.2461,Y 7.4826,Z 56,A -2.0928,B 0,C 0,E1 0.1598,E2 -629.9276} C_DIS
LIN {X 7.196,Y 6.5745,Z 56,A -2.0964,B 0,C 0,E1 0.1598,E2 -629.9277} C_DIS
LIN {X 8.0129,Y 5.5491,Z 56,A -2.1099,B 0,C 0,E1 0.1598,E2 -629.9279} C_DIS
LIN {X 8.657,Y 4.4793,Z 56,A -2.1317,B 0,C 0,E1 0.1598,E2 -629.9281} C_DIS
LIN {X 9.0607,Y 3.5934,Z 56,A -2.155,B 0,C 0,E1 0.1598,E2 -629.9278} C_DIS
LIN {X 9.4604,Y 2.3472,Z 56,A -2.1932,B 0,C 0,E1 0.1598,E2 -629.9282} C_DIS
LIN {X 9.6548,Y 1.3388,Z 56,A -2.2294,B 0,C 0,E1 0.1598,E2 -629.928} C_DIS
LIN {X 9.7428,Y 0.2908,Z 56,A -2.271,B 0,C 0,E1 0.1598,E2 -629.928} C_DIS
LIN {X 9.7083,Y -0.8677,Z 56,A -2.3218,B 0,C 0,E1 0.1598,E2 -629.9283} C_DIS
LIN {X 9.5298,Y -2.0308,Z 56,A -2.3781,B 0,C 0,E1 0.1598,E2 -629.9284} C_DIS
LIN {X 9.1557,Y -3.3436,Z 56,A -2.4478,B 0,C 0,E1 0.1598,E2 -629.9287} C_DIS
LIN {X 8.6369,Y -4.5175,Z 56,A -2.5172,B 0,C 0,E1 0.1598,E2 -629.9287} C_DIS
LIN {X 7.9253,Y -5.6742,Z 56,A -2.5931,B 0,C 0,E1 0.1598,E2 -629.9286} C_DIS
LIN {X 7.4658,Y -6.2667,Z 56,A -2.6357,B 0,C 0,E1 0.1598,E2 -629.9282} C_DIS
LIN {X 6.8092,Y -6.9745,Z 56,A -2.6901,B 0,C 0,E1 0.1598,E2 -629.9282} C_DIS
LIN {X 6.0649,Y -7.6303,Z 56,A -2.7455,B 0,C 0,E1 0.1598,E2 -629.9282} C_DIS
LIN {X 4.466,Y -8.6637,Z 56,A -2.8482,B 0,C 0,E1 0.1598,E2 -629.9285} C_DIS
LIN {X 3.7053,Y -9.0148,Z 56,A -2.8913,B 0,C 0,E1 0.1598,E2 -629.9283} C_DIS
LIN {X 2.2968,Y -9.4727,Z 56,A -2.9624,B 0,C 0,E1 0.1598,E2 -629.9285} C_DIS
LIN {X 1.0187,Y -9.6937,Z 56,A -3.0187,B 0,C 0,E1 0.1598,E2 -629.9285} C_DIS
LIN {X 0.0339,Y -9.7462,Z 56,A -3.0571,B 0,C 0,E1 0.1598,E2 -629.9285} C_DIS
Enddeposition()
LIN {X 0.0339,Y -9.7462,Z 56,A -3.0571,B 0,C 0,E1 0.1598,E2 -629.9285} C_DIS
Startdeposition()
$VEL.CP = VEL_PRINT
LIN {X 0.5104,Y -8.7341,Z 56,A -2.9955,B 0,C 0,E1 0.1598,E2 -629.9291} C_DIS
LIN {X 1.4828,Y -8.6227,Z 56,A -2.9557,B 0,C 0,E1 0.1598,E2 -629.9284} C_DIS
LIN {X 2.7384,Y -8.3092,Z 56,A -2.8963,B 0,C 0,E1 0.1598,E2 -629.9284} C_DIS
LIN {X 4.0371,Y -7.7619,Z 56,A -2.8253,B 0,C 0,E1 0.1598,E2 -629.9284} C_DIS
LIN {X 5.5518,Y -6.7619,Z 56,A -2.7266,B 0,C 0,E1 0.1598,E2 -629.9286} C_DIS
LIN {X 6.5759,Y -5.771,Z 56,A -2.6464,B 0,C 0,E1 0.1598,E2 -629.9287} C_DIS
LIN {X 7.5561,Y -4.4101,Z 56,A -2.552,B 0,C 0,E1 0.1598,E2 -629.9287} C_DIS
LIN {X 8.1566,Y -3.1646,Z 56,A -2.4767,B 0,C 0,E1 0.1598,E2 -629.9287} C_DIS
LIN {X 8.4561,Y -2.2347,Z 56,A -2.4263,B 0,C 0,E1 0.1598,E2 -629.9281} C_DIS
LIN {X 8.6212,Y -1.4707,Z 56,A -2.3876,B 0,C 0,E1 0.1598,E2 -629.928} C_DIS
LIN {X 8.7475,Y -0.0949,Z 56,A -2.3233,B 0,C 0,E1 0.1598,E2 -629.9287} C_DIS
LIN {X 8.6095,Y 1.5556,Z 56,A -2.2574,B 0,C 0,E1 0.1598,E2 -629.929} C_DIS
LIN {X 8.3328,Y 2.6603,Z 56,A -2.2211,B 0,C 0,E1 0.1598,E2 -629.9281} C_DIS
LIN {X 8.1006,Y 3.2992,Z 56,A -2.2028,B 0,C 0,E1 0.1598,E2 -629.9276} C_DIS
LIN {X 7.6308,Y 4.2802,Z 56,A -2.1779,B 0,C 0,E1 0.1598,E2 -629.9279} C_DIS
LIN {X 6.8757,Y 5.4093,Z 56,A -2.1572,B 0,C 0,E1 0.1598,E2 -629.9282} C_DIS
LIN {X 6.0869,Y 6.2842,Z 56,A -2.1493,B 0,C 0,E1 0.1598,E2 -629.9278} C_DIS
LIN {X 5.2669,Y 6.9862,Z 56,A -2.1498,B 0,C 0,E1 0.1598,E2 -629.9276} C_DIS
LIN {X 4.111,Y 7.7232,Z 56,A -2.161,B 0,C 0,E1 0.1598,E2 -629.9276} C_DIS
LIN {X 2.9733,Y 8.2246,Z 56,A -2.1819,B 0,C 0,E1 0.1598,E2 -629.9276} C_DIS
LIN {X 1.8672,Y 8.5476,Z 56,A -2.2091,B 0,C 0,E1 0.1598,E2 -629.9275} C_DIS
LIN {X 1.0911,Y 8.6809,Z 56,A -2.2321,B 0,C 0,E1 0.1598,E2 -629.9275} C_DIS
LIN {X -0.142,Y 8.7479,Z 56,A -2.2748,B 0,C 0,E1 0.1598,E2 -629.9275} C_DIS
LIN {X -1.3336,Y 8.647,Z 56,A -2.3231,B 0,C 0,E1 0.1598,E2 -629.9275} C_DIS
LIN {X -2.4831,Y 8.3892,Z 56,A -2.3764,B 0,C 0,E1 0.1598,E2 -629.9276} C_DIS
LIN {X -3.6077,Y 7.9705,Z 56,A -2.4357,B 0,C 0,E1 0.1598,E2 -629.9278} C_DIS
LIN {X -4.5071,Y 7.4948,Z 56,A -2.489,B 0,C 0,E1 0.1598,E2 -629.9278} C_DIS
LIN {X -5.8079,Y 6.5436,Z 56,A -2.5769,B 0,C 0,E1 0.1598,E2 -629.9284} C_DIS
LIN {X -6.778,Y 5.5324,Z 56,A -2.6556,B 0,C 0,E1 0.1598,E2 -629.9284} C_DIS
LIN {X -7.7037,Y 4.1465,Z 56,A -2.7479,B 0,C 0,E1 0.1598,E2 -629.929} C_DIS
LIN {X -8.2773,Y 2.8339,Z 56,A -2.8245,B 0,C 0,E1 0.1598,E2 -629.9292} C_DIS
LIN {X -8.6412,Y 1.3711,Z 56,A -2.8997,B 0,C 0,E1 0.1598,E2 -629.9295} C_DIS
LIN {X -8.7442,Y 0.129,Z 56,A -2.9564,B 0,C 0,E1 0.1598,E2 -629.9292} C_DIS
LIN {X -8.7175,Y -0.6802,Z 56,A -2.9902,B 0,C 0,E1 0.1598,E2 -629.9288} C_DIS
LIN {X -8.618,Y -1.4836,Z 56,A -3.0206,B 0,C 0,E1 0.1598,E2 -629.9288} C_DIS
LIN {X -8.3468,Y -2.6224,Z 56,A -3.0586,B 0,C 0,E1 0.1598,E2 -629.9292} C_DIS
LIN {X -7.9085,Y -3.7426,Z 56,A -3.0901,B 0,C 0,E1 0.1598,E2 -629.9292} C_DIS
LIN {X -7.3385,Y -4.7639,Z 56,A -3.1125,B 0,C 0,E1 0.1598,E2 -629.9292} C_DIS
LIN {X -6.6355,Y -5.7026,Z 56,A -3.1267,B 0,C 0,E1 0.1598,E2 -629.9291} C_DIS
LIN {X -5.993,Y -6.3742,Z 56,A -3.1318,B 0,C 0,E1 0.1598,E2 -629.9289} C_DIS
LIN {X -5.0811,Y -7.1224,Z 56,A -3.1302,B 0,C 0,E1 0.1598,E2 -629.9289} C_DIS
LIN {X -3.9529,Y -7.8046,Z 56,A -3.1179,B 0,C 0,E1 0.1598,E2 -629.9289} C_DIS
LIN {X -2.9362,Y -8.2419,Z 56,A -3.0994,B 0,C 0,E1 0.1598,E2 -629.9287} C_DIS
LIN {X -1.6239,Y -8.5972,Z 56,A -3.0665,B 0,C 0,E1 0.1598,E2 -629.9286} C_DIS
LIN {X -0.5816,Y -8.7297,Z 56,A -3.034,B 0,C 0,E1 0.1598,E2 -629.9285} C_DIS
LIN {X -0.5816,Y -8.7297,Z 56,A -3.034,B 0,C 0,E1 0.1598,E2 -629.9285} C_DIS
Enddeposition()
LIN {X -0.0322,Y -7.7512,Z 56,A -2.9706,B 0,C 0,E1 0.1598,E2 -629.9298} C_DIS
Startdeposition()
$VEL.CP = VEL_PRINT
LIN {X -1.4492,Y -7.6146,Z 56,A -3.018,B 0,C 0,E1 0.1598,E2 -629.9285} C_DIS
LIN {X -2.3127,Y -7.3957,Z 56,A -3.0403,B 0,C 0,E1 0.1598,E2 -629.9285} C_DIS
LIN {X -3.3298,Y -6.9995,Z 56,A -3.0607,B 0,C 0,E1 0.1598,E2 -629.9286} C_DIS
LIN {X -4.477,Y -6.3277,Z 56,A -3.074,B 0,C 0,E1 0.1598,E2 -629.9288} C_DIS
LIN {X -5.2921,Y -5.6634,Z 56,A -3.0757,B 0,C 0,E1 0.1598,E2 -629.9288} C_DIS
LIN {X -6.2189,Y -4.6267,Z 56,A -3.0652,B 0,C 0,E1 0.1598,E2 -629.9292} C_DIS
LIN {X -6.7515,Y -3.8078,Z 56,A -3.0503,B 0,C 0,E1 0.1598,E2 -629.9288} C_DIS
LIN {X -7.2253,Y -2.7949,Z 56,A -3.0244,B 0,C 0,E1 0.1598,E2 -629.9291} C_DIS
LIN {X -7.4764,Y -2.0271,Z 56,A -3.0013,B 0,C 0,E1 0.1598,E2 -629.9288} C_DIS
LIN {X -7.6476,Y -1.2376,Z 56,A -2.9741,B 0,C 0,E1 0.1598,E2 -629.9288} C_DIS
LIN {X -7.7356,Y -0.4345,Z 56,A -2.9433,B 0,C 0,E1 0.1598,E2 -629.9287} C_DIS
LIN {X -7.7181,Y 0.7146,Z 56,A -2.8936,B 0,C 0,E1 0.1598,E2 -629.929} C_DIS
LIN {X -7.5348,Y 1.8006,Z 56,A -2.8409,B 0,C 0,E1 0.1598,E2 -629.9289} C_DIS
LIN {X -7.2514,Y 2.7377,Z 56,A -2.7908,B 0,C 0,E1 0.1598,E2 -629.9287} C_DIS
LIN {X -6.6937,Y 3.9086,Z 56,A -2.7204,B 0,C 0,E1 0.1598,E2 -629.9288} C_DIS
LIN {X -6.0845,Y 4.802,Z 56,A -2.6604,B 0,C 0,E1 0.1598,E2 -629.9284} C_DIS
LIN {X -5.2437,Y 5.7037,Z 56,A -2.5912,B 0,C 0,E1 0.1598,E2 -629.9284} C_DIS
LIN {X -4.6045,Y 6.2287,Z 56,A -2.5456,B 0,C 0,E1 0.1598,E2 -629.928} C_DIS
LIN {X -3.7367,Y 6.7908,Z 56,A -2.4898,B 0,C 0,E1 0.1598,E2 -629.928} C_DIS
LIN {X -2.6869,Y 7.2704,Z 56,A -2.4308,B 0,C 0,E1 0.1598,E2 -629.9278} C_DIS
LIN {X -1.6382,Y 7.5761,Z 56,A -2.3791,B 0,C 0,E1 0.1598,E2 -629.9276} C_DIS
LIN {X -0.7261,Y 7.7133,Z 56,A -2.3397,B 0,C 0,E1 0.1598,E2 -629.9276} C_DIS
LIN {X 0.0111,Y 7.7457,Z 56,A -2.3111,B 0,C 0,E1 0.1598,E2 -629.9276} C_DIS
LIN {X 0.7482,Y 7.7118,Z 56,A -2.2853,B 0,C 0,E1 0.1598,E2 -629.9275} C_DIS
LIN {X 1.4786,Y 7.6061,Z 56,A -2.2629,B 0,C 0,E1 0.1598,E2 -629.9275} C_DIS
LIN {X 2.5368,Y 7.3241,Z 56,A -2.2358,B 0,C 0,E1 0.1598,E2 -629.9275} C_DIS
LIN {X 3.4522,Y 6.9399,Z 56,A -2.2183,B 0,C 0,E1 0.1598,E2 -629.9275} C_DIS
LIN {X 4.4053,Y 6.3776,Z 56,A -2.207,B 0,C 0,E1 0.1598,E2 -629.9275} C_DIS
LIN {X 5.2204,Y 5.7265,Z 56,A -2.2046,B 0,C 0,E1 0.1598,E2 -629.9276} C_DIS
LIN {X 5.6722,Y 5.2793,Z 56,A -2.2072,B 0,C 0,E1 0.1598,E2 -629.9276} C_DIS
LIN {X 6.312,Y 4.499,Z 56,A -2.2166,B 0,C 0,E1 0.1598,E2 -629.9278} C_DIS
LIN {X 6.8251,Y 3.6743,Z 56,A -2.2329,B 0,C 0,E1 0.1598,E2 -629.9278} C_DIS
LIN {X 7.2768,Y 2.6697,Z 56,A -2.259,B 0,C 0,E1 0.1598,E2 -629.928} C_DIS
LIN {X 7.5138,Y 1.9039,Z 56,A -2.2832,B 0,C 0,E1 0.1598,E2 -629.9278} C_DIS
LIN {X 7.726,Y 0.623,Z 56,A -2.3296,B 0,C 0,E1 0.1598,E2 -629.9284} C_DIS
LIN {X 7.735,Y -0.4981,Z 56,A -2.3774,B 0,C 0,E1 0.1598,E2 -629.9284} C_DIS
LIN {X 7.5905,Y -1.5693,Z 56,A -2.4286,B 0,C 0,E1 0.1598,E2 -629.9284} C_DIS
LIN {X 7.212,Y -2.8402,Z 56,A -2.4965,B 0,C 0,E1 0.1598,E2 -629.9287} C_DIS
LIN {X 6.5667,Y -4.1182,Z 56,A -2.5747,B 0,C 0,E1 0.1598,E2 -629.929} C_DIS
LIN {X 5.6593,Y -5.2962,Z 56,A -2.6588,B 0,C 0,E1 0.1598,E2 -629.9287} C_DIS
LIN {X 4.1767,Y -6.5293,Z 56,A -2.7659,B 0,C 0,E1 0.1598,E2 -629.9289} C_DIS
LIN {X 3.2239,Y -7.048,Z 56,A -2.8235,B 0,C 0,E1 0.1598,E2 -629.9284} C_DIS
LIN {X 1.9416,Y -7.5041,Z 56,A -2.8901,B 0,C 0,E1 0.1598,E2 -629.9284} C_DIS
LIN {X -0.0322,Y -7.7512,Z 56,A -2.973,B 0,C 0,E1 0.1598,E2 -629.9284} C_DIS
Enddeposition()
LIN {X -0.0322,Y -7.7512,Z 56,A -2.973,B 0,C 0,E1 0.1598,E2 -629.9284} C_DIS
Startdeposition()
$VEL.CP = VEL_PRINT
LIN {X 0.4901,Y -6.7353,Z 56,A -2.9097,B 0,C 0,E1 0.1598,E2 -629.929} C_DIS
LIN {X 1.6074,Y -6.5542,Z 56,A -2.8616,B 0,C 0,E1 0.1598,E2 -629.9283} C_DIS
LIN {X 2.3912,Y -6.3113,Z 56,A -2.8225,B 0,C 0,E1 0.1598,E2 -629.9283} C_DIS
LIN {X 3.1389,Y -5.9736,Z 56,A -2.7806,B 0,C 0,E1 0.1598,E2 -629.9282} C_DIS
LIN {X 4.3182,Y -5.1923,Z 56,A -2.7037,B 0,C 0,E1 0.1598,E2 -629.9284} C_DIS
LIN {X 5.3098,Y -4.1669,Z 56,A -2.6233,B 0,C 0,E1 0.1598,E2 -629.9284} C_DIS
LIN {X 5.8446,Y -3.3823,Z 56,A -2.5701,B 0,C 0,E1 0.1598,E2 -629.9284} C_DIS
LIN {X 6.4124,Y -2.1154,Z 56,A -2.4947,B 0,C 0,E1 0.1598,E2 -629.9287} C_DIS
LIN {X 6.7192,Y -0.6766,Z 56,A -2.4218,B 0,C 0,E1 0.1598,E2 -629.9287} C_DIS
LIN {X 6.7213,Y 0.654,Z 56,A -2.3649,B 0,C 0,E1 0.1598,E2 -629.9285} C_DIS
LIN {X 6.5555,Y 1.5974,Z 56,A -2.3312,B 0,C 0,E1 0.1598,E2 -629.928} C_DIS
LIN {X 6.334,Y 2.3308,Z 56,A -2.3082,B 0,C 0,E1 0.1598,E2 -629.9278} C_DIS
LIN {X 6.0282,Y 3.0332,Z 56,A -2.2895,B 0,C 0,E1 0.1598,E2 -629.9278} C_DIS
LIN {X 5.6454,Y 3.6969,Z 56,A -2.2753,B 0,C 0,E1 0.1598,E2 -629.9278} C_DIS
LIN {X 5.189,Y 4.3123,Z 56,A -2.2659,B 0,C 0,E1 0.1598,E2 -629.9277} C_DIS
LIN {X 4.6674,Y 4.8733,Z 56,A -2.2612,B 0,C 0,E1 0.1598,E2 -629.9277} C_DIS
LIN {X 3.8253,Y 5.5653,Z 56,A -2.2626,B 0,C 0,E1 0.1598,E2 -629.9277} C_DIS
LIN {X 2.8745,Y 6.1109,Z 56,A -2.2746,B 0,C 0,E1 0.1598,E2 -629.9277} C_DIS
LIN {X 1.8895,Y 6.4797,Z 56,A -2.2953,B 0,C 0,E1 0.1598,E2 -629.9276} C_DIS
LIN {X 1.2397,Y 6.6342,Z 56,A -2.3128,B 0,C 0,E1 0.1598,E2 -629.9276} C_DIS
LIN {X 0.0967,Y 6.7525,Z 56,A -2.3499,B 0,C 0,E1 0.1598,E2 -629.9276} C_DIS
LIN {X -1.3484,Y 6.6119,Z 56,A -2.4092,B 0,C 0,E1 0.1598,E2 -629.9276} C_DIS
LIN {X -2.5251,Y 6.2634,Z 56,A -2.4674,B 0,C 0,E1 0.1598,E2 -629.9278} C_DIS
LIN {X -3.4681,Y 5.7948,Z 56,A -2.522,B 0,C 0,E1 0.1598,E2 -629.9278} C_DIS
LIN {X -4.4072,Y 5.117,Z 56,A -2.5852,B 0,C 0,E1 0.1598,E2 -629.9281} C_DIS
LIN {X -5.1166,Y 4.4022,Z 56,A -2.6417,B 0,C 0,E1 0.1598,E2 -629.9281} C_DIS
LIN {X -5.6038,Y 3.7606,Z 56,A -2.6869,B 0,C 0,E1 0.1598,E2 -629.9282} C_DIS
LIN {X -6.105,Y 2.8872,Z 56,A -2.7421,B 0,C 0,E1 0.1598,E2 -629.9285} C_DIS
LIN {X -6.4452,Y 2.0156,Z 56,A -2.7917,B 0,C 0,E1 0.1598,E2 -629.9285} C_DIS
LIN {X -6.6947,Y 0.8512,Z 56,A -2.8498,B 0,C 0,E1 0.1598,E2 -629.929} C_DIS
LIN {X -6.751,Y 0.1759,Z 56,A -2.8811,B 0,C 0,E1 0.1598,E2 -629.9285} C_DIS
LIN {X -6.6956,Y -0.8544,Z 56,A -2.9224,B 0,C 0,E1 0.1598,E2 -629.9289} C_DIS
LIN {X -6.5828,Y -1.4876,Z 56,A -2.9454,B 0,C 0,E1 0.1598,E2 -629.9286} C_DIS
LIN {X -6.2662,Y -2.5182,Z 56,A -2.9772,B 0,C 0,E1 0.1598,E2 -629.929} C_DIS
LIN {X -5.7492,Y -3.543,Z 56,A -3.0018,B 0,C 0,E1 0.1598,E2 -629.929} C_DIS
LIN {X -5.1515,Y -4.3666,Z 56,A -3.015,B 0,C 0,E1 0.1598,E2 -629.9288} C_DIS
LIN {X -3.9556,Y -5.4735,Z 56,A -3.0179,B 0,C 0,E1 0.1598,E2 -629.9291} C_DIS
LIN {X -3.0854,Y -6.0025,Z 56,A -3.0089,B 0,C 0,E1 0.1598,E2 -629.9286} C_DIS
LIN {X -2.0235,Y -6.4427,Z 56,A -2.9888,B 0,C 0,E1 0.1598,E2 -629.9286} C_DIS
LIN {X -0.6386,Y -6.7178,Z 56,A -2.9498,B 0,C 0,E1 0.1598,E2 -629.9284} C_DIS
LIN {X -0.6386,Y -6.7178,Z 56,A -2.9498,B 0,C 0,E1 0.1598,E2 -629.9284} C_DIS
Enddeposition()
LIN {X -0.0086,Y -5.7552,Z 56,A -2.8841,B 0,C 0,E1 0.1598,E2 -629.9297} C_DIS
Startdeposition()
$VEL.CP = VEL_PRINT
LIN {X -1.1481,Y -5.6395,Z 56,A -2.9223,B 0,C 0,E1 0.1598,E2 -629.9284} C_DIS
LIN {X -2.4148,Y -5.2242,Z 56,A -2.9511,B 0,C 0,E1 0.1598,E2 -629.9284} C_DIS
LIN {X -3.3337,Y -4.6914,Z 56,A -2.962,B 0,C 0,E1 0.1598,E2 -629.9285} C_DIS
LIN {X -3.9595,Y -4.1765,Z 56,A -2.9631,B 0,C 0,E1 0.1598,E2 -629.9285} C_DIS
LIN {X -4.9566,Y -2.925,Z 56,A -2.9458,B 0,C 0,E1 0.1598,E2 -629.9293} C_DIS
LIN {X -5.5802,Y -1.4087,Z 56,A -2.904,B 0,C 0,E1 0.1598,E2 -629.9295} C_DIS
LIN {X -5.7259,Y -0.5386,Z 56,A -2.8732,B 0,C 0,E1 0.1598,E2 -629.9287} C_DIS
LIN {X -5.7467,Y 0.1668,Z 56,A -2.8441,B 0,C 0,E1 0.1598,E2 -629.9285} C_DIS
LIN {X -5.6845,Y 0.8697,Z 56,A -2.812,B 0,C 0,E1 0.1598,E2 -629.9285} C_DIS
LIN {X -5.5357,Y 1.5596,Z 56,A -2.7773,B 0,C 0,E1 0.1598,E2 -629.9284} C_DIS
LIN {X -5.3022,Y 2.2257,Z 56,A -2.7405,B 0,C 0,E1 0.1598,E2 -629.9284} C_DIS
LIN {X -4.9887,Y 2.8578,Z 56,A -2.7021,B 0,C 0,E1 0.1598,E2 -629.9282} C_DIS
LIN {X -4.6012,Y 3.4475,Z 56,A -2.6628,B 0,C 0,E1 0.1598,E2 -629.9282} C_DIS
LIN {X -4.1461,Y 3.987,Z 56,A -2.6232,B 0,C 0,E1 0.1598,E2 -629.9281} C_DIS
LIN {X -3.6258,Y 4.464,Z 56,A -2.5838,B 0,C 0,E1 0.1598,E2 -629.928} C_DIS
LIN {X -3.0514,Y 4.8739,Z 56,A -2.5453,B 0,C 0,E1 0.1598,E2 -629.928} C_DIS
LIN {X -2.431,Y 5.2104,Z 56,A -2.5082,B 0,C 0,E1 0.1598,E2 -629.9278} C_DIS
LIN {X -1.7751,Y 5.4708,Z 56,A -2.4729,B 0,C 0,E1 0.1598,E2 -629.9278} C_DIS
LIN {X -1.0913,Y 5.645,Z 56,A -2.4403,B 0,C 0,E1 0.1598,E2 -629.9277} C_DIS
LIN {X -0.3916,Y 5.7366,Z 56,A -2.4107,B 0,C 0,E1 0.1598,E2 -629.9277} C_DIS
LIN {X 0.4906,Y 5.7341,Z 56,A -2.3782,B 0,C 0,E1 0.1598,E2 -629.9277} C_DIS
LIN {X 1.7022,Y 5.4975,Z 56,A -2.3436,B 0,C 0,E1 0.1598,E2 -629.9277} C_DIS
LIN {X 2.2804,Y 5.2788,Z 56,A -2.3316,B 0,C 0,E1 0.1598,E2 -629.9276} C_DIS
LIN {X 3.01,Y 4.897,Z 56,A -2.3209,B 0,C 0,E1 0.1598,E2 -629.9276} C_DIS
LIN {X 3.6797,Y 4.4179,Z 56,A -2.3166,B 0,C 0,E1 0.1598,E2 -629.9276} C_DIS
LIN {X 4.2728,Y 3.8469,Z 56,A -2.319,B 0,C 0,E1 0.1598,E2 -629.9277} C_DIS
LIN {X 4.777,Y 3.196,Z 56,A -2.3281,B 0,C 0,E1 0.1598,E2 -629.9277} C_DIS
LIN {X 5.1845,Y 2.4808,Z 56,A -2.3436,B 0,C 0,E1 0.1598,E2 -629.9279} C_DIS
LIN {X 5.4886,Y 1.7157,Z 56,A -2.365,B 0,C 0,E1 0.1598,E2 -629.9279} C_DIS
LIN {X 5.6765,Y 0.914,Z 56,A -2.3923,B 0,C 0,E1 0.1598,E2 -629.9279} C_DIS
LIN {X 5.75,Y -0.2449,Z 56,A -2.4387,B 0,C 0,E1 0.1598,E2 -629.9284} C_DIS
LIN {X 5.6272,Y -1.1824,Z 56,A -2.4835,B 0,C 0,E1 0.1598,E2 -629.9282} C_DIS
LIN {X 5.4233,Y -1.911,Z 56,A -2.5223,B 0,C 0,E1 0.1598,E2 -629.9281} C_DIS
LIN {X 5.0415,Y -2.7761,Z 56,A -2.5731,B 0,C 0,E1 0.1598,E2 -629.9283} C_DIS
LIN {X 4.4531,Y -3.6459,Z 56,A -2.632,B 0,C 0,E1 0.1598,E2 -629.9283} C_DIS
LIN {X 3.6827,Y -4.4227,Z 56,A -2.6935,B 0,C 0,E1 0.1598,E2 -629.9283} C_DIS
LIN {X 3.0817,Y -4.8588,Z 56,A -2.7343,B 0,C 0,E1 0.1598,E2 -629.9283} C_DIS
LIN {X 2.3761,Y -5.2388,Z 56,A -2.7765,B 0,C 0,E1 0.1598,E2 -629.9282} C_DIS
LIN {X 1.5588,Y -5.54,Z 56,A -2.8194,B 0,C 0,E1 0.1598,E2 -629.9282} C_DIS
LIN {X 0.7047,Y -5.7113,Z 56,A -2.8581,B 0,C 0,E1 0.1598,E2 -629.9282} C_DIS
LIN {X -0.0086,Y -5.7552,Z 56,A -2.8861,B 0,C 0,E1 0.1598,E2 -629.9282} C_DIS
Enddeposition()
LIN {X -0.0086,Y -5.7552,Z 56,A -2.8861,B 0,C 0,E1 0.1598,E2 -629.9282} C_DIS
Startdeposition()
$VEL.CP = VEL_PRINT
LIN {X 0.3786,Y -4.7407,Z 56,A -2.8278,B 0,C 0,E1 0.1598,E2 -629.9289} C_DIS
LIN {X 1.0239,Y -4.6443,Z 56,A -2.8007,B 0,C 0,E1 0.1598,E2 -629.9282} C_DIS
LIN {X 1.6498,Y -4.4603,Z 56,A -2.7699,B 0,C 0,E1 0.1598,E2 -629.9282} C_DIS
LIN {X 2.2445,Y -4.1922,Z 56,A -2.7366,B 0,C 0,E1 0.1598,E2 -629.9282} C_DIS
LIN {X 2.7966,Y -3.8449,Z 56,A -2.7015,B 0,C 0,E1 0.1598,E2 -629.9281} C_DIS
LIN {X 3.4135,Y -3.3121,Z 56,A -2.656,B 0,C 0,E1 0.1598,E2 -629.9281} C_DIS
LIN {X 3.9286,Y -2.6804,Z 56,A -2.61,B 0,C 0,E1 0.1598,E2 -629.9281} C_DIS
LIN {X 4.2582,Y -2.1174,Z 56,A -2.5739,B 0,C 0,E1 0.1598,E2 -629.9281} C_DIS
LIN {X 4.5579,Y -1.3594,Z 56,A -2.5304,B 0,C 0,E1 0.1598,E2 -629.9281} C_DIS
LIN {X 4.7218,Y -0.5609,Z 56,A -2.4903,B 0,C 0,E1 0.1598,E2 -629.9281} C_DIS
LIN {X 4.7533,Y 0.1723,Z 56,A -2.4578,B 0,C 0,E1 0.1598,E2 -629.9281} C_DIS
LIN {X 4.6531,Y 0.9813,Z 56,A -2.4269,B 0,C 0,E1 0.1598,E2 -629.9281} C_DIS
LIN {X 4.3873,Y 1.8375,Z 56,A -2.4001,B 0,C 0,E1 0.1598,E2 -629.9281} C_DIS
LIN {X 4.0093,Y 2.5597,Z 56,A -2.3833,B 0,C 0,E1 0.1598,E2 -629.9279} C_DIS
LIN {X 3.5127,Y 3.2062,Z 56,A -2.3741,B 0,C 0,E1 0.1598,E2 -629.9279} C_DIS
LIN {X 2.9131,Y 3.7582,Z 56,A -2.3727,B 0,C 0,E1 0.1598,E2 -629.9278} C_DIS
LIN {X 2.2333,Y 4.1995,Z 56,A -2.379,B 0,C 0,E1 0.1598,E2 -629.9278} C_DIS
LIN {X 1.6172,Y 4.4731,Z 56,A -2.3902,B 0,C 0,E1 0.1598,E2 -629.9277} C_DIS
LIN {X 0.8579,Y 4.677,Z 56,A -2.4095,B 0,C 0,E1 0.1598,E2 -629.9277} C_DIS
LIN {X 0.188,Y 4.7507,Z 56,A -2.4311,B 0,C 0,E1 0.1598,E2 -629.9277} C_DIS
LIN {X -0.4856,Y 4.7297,Z 56,A -2.4568,B 0,C 0,E1 0.1598,E2 -629.9277} C_DIS
LIN {X -1.1494,Y 4.6135,Z 56,A -2.4862,B 0,C 0,E1 0.1598,E2 -629.9277} C_DIS
LIN {X -1.7902,Y 4.4047,Z 56,A -2.5187,B 0,C 0,E1 0.1598,E2 -629.9278} C_DIS
LIN {X -2.492,Y 4.0508,Z 56,A -2.5595,B 0,C 0,E1 0.1598,E2 -629.9278} C_DIS
LIN {X -3.1245,Y 3.584,Z 56,A -2.6026,B 0,C 0,E1 0.1598,E2 -629.928} C_DIS
LIN {X -3.6001,Y 3.1064,Z 56,A -2.6404,B 0,C 0,E1 0.1598,E2 -629.928} C_DIS
LIN {X -4.003,Y 2.5663,Z 56,A -2.6781,B 0,C 0,E1 0.1598,E2 -629.9282} C_DIS
LIN {X -4.3703,Y 1.8713,Z 56,A -2.7211,B 0,C 0,E1 0.1598,E2 -629.9282} C_DIS
LIN {X -4.5922,Y 1.2349,Z 56,A -2.7563,B 0,C 0,E1 0.1598,E2 -629.9283} C_DIS
LIN {X -4.7198,Y 0.5731,Z 56,A -2.789,B 0,C 0,E1 0.1598,E2 -629.9283} C_DIS
LIN {X -4.7458,Y -0.3286,Z 56,A -2.828,B 0,C 0,E1 0.1598,E2 -629.9287} C_DIS
LIN {X -4.6075,Y -1.1676,Z 56,A -2.8587,B 0,C 0,E1 0.1598,E2 -629.9286} C_DIS
LIN {X -4.3931,Y -1.8132,Z 56,A -2.8784,B 0,C 0,E1 0.1598,E2 -629.9285} C_DIS
LIN {X -4.0886,Y -2.4214,Z 56,A -2.8931,B 0,C 0,E1 0.1598,E2 -629.9285} C_DIS
LIN {X -3.7009,Y -2.9801,Z 56,A -2.9026,B 0,C 0,E1 0.1598,E2 -629.9285} C_DIS
LIN {X -3.2369,Y -3.4773,Z 56,A -2.9067,B 0,C 0,E1 0.1598,E2 -629.9285} C_DIS
LIN {X -2.708,Y -3.9047,Z 56,A -2.9055,B 0,C 0,E1 0.1598,E2 -629.9285} C_DIS
LIN {X -2.123,Y -4.2519,Z 56,A -2.8989,B 0,C 0,E1 0.1598,E2 -629.9284} C_DIS
LIN {X -1.494,Y -4.5109,Z 56,A -2.8868,B 0,C 0,E1 0.1598,E2 -629.9284} C_DIS
LIN {X -0.8349,Y -4.679,Z 56,A -2.8698,B 0,C 0,E1 0.1598,E2 -629.9283} C_DIS
LIN {X 0.0118,Y -4.7573,Z 56,A -2.8421,B 0,C 0,E1 0.1598,E2 -629.9283} C_DIS
Enddeposition()
LIN {X 0.0118,Y -4.7573,Z 61,A -2.8318,B 0,C 0,E1 0.1598,E2 -629.928} C_DIS
LIN {X 0.0118,Y -4.7572,Z 76,A -2.8054,B 0,C 0,E1 0.1598,E2 -629.9269} C_DIS
LIN {X 0.0118,Y -4.7572,Z 95.1262,A -2.7798,B 0,C 0,E1 0.1598,E2 -629.9267} C_DIS
LIN {X -0.035,Y -34.947,Z 95.1262,A -97.4394,B 24.8325,C -2.9854,E1 24.9993,E2 -540.0022} C_DIS
LIN {X -0.035,Y -34.947,Z 75.1262,A -97.1108,B 24.8477,C -2.8474,E1 24.9993,E2 -540.0022} C_DIS
LIN {X 0.0049,Y -28.6078,Z 61.5315,A -97.1498,B 24.8459,C -2.8637,E1 24.9993,E2 -540.0022} C_DIS
LIN {X 0.0182,Y -26.4948,Z 57,A -97.1642,B 24.8453,C -2.8698,E1 24.9993,E2 -540.0022} C_DIS
Startdeposition()
$VEL.CP = VEL_PRINT
LIN {X -1.6249,Y -26.4483,Z 57,A -101.348,B 24.8459,C -2.8639,E1 24.9876,E2 -535.8034} C_DIS
LIN {X -3.5662,Y -26.2577,Z 57,A -105.5489,B 24.8459,C -2.8646,E1 24.9759,E2 -531.6014} C_DIS
LIN {X -5.4378,Y -25.9348,Z 57,A -109.6692,B 24.8457,C -2.8659,E1 24.9646,E2 -527.4798} C_DIS
LIN {X -7.2913,Y -25.4758,Z 57,A -113.8197,B 24.8454,C -2.8682,E1 24.9534,E2 -523.3284} C_DIS
LIN {X -9.1275,Y -24.877,Z 57,A -117.997,B 24.8451,C -2.8715,E1 24.9424,E2 -519.1512} C_DIS
LIN {X -10.9573,Y -24.1271,Z 57,A -122.2623,B 24.8446,C -2.876,E1 24.9315,E2 -514.8865} C_DIS
LIN {X -12.6608,Y -23.2783,Z 57,A -126.4266,B 24.8441,C -2.8808,E1 24.9212,E2 -510.7221} C_DIS
LIN {X -14.358,Y -22.2716,Z 57,A -130.7477,B 24.8434,C -2.8866,E1 24.9109,E2 -506.4013} C_DIS
LIN {X -16.0303,Y -21.1003,Z 57,A -135.1721,B 24.8427,C -2.8938,E1 24.9009,E2 -501.9786} C_DIS
LIN {X -17.481,Y -19.9146,Z 57,A -139.1752,B 24.8418,C -2.9016,E1 24.8924,E2 -497.9788} C_DIS
LIN {X -18.8729,Y -18.6007,Z 57,A -143.3924,B 24.8409,C -2.9095,E1 24.884,E2 -493.7627} C_DIS
LIN {X -20.2401,Y -17.1033,Z 57,A -147.8172,B 24.8399,C -2.9188,E1 24.8758,E2 -489.3403} C_DIS
LIN {X -21.4101,Y -15.6135,Z 57,A -151.9315,B 24.8389,C -2.9283,E1 24.8689,E2 -485.2291} C_DIS
LIN {X -22.5391,Y -13.9348,Z 57,A -156.3311,B 24.8377,C -2.9391,E1 24.8623,E2 -480.8331} C_DIS
LIN {X -23.5214,Y -12.2037,Z 57,A -160.6499,B 24.8364,C -2.9504,E1 24.8565,E2 -476.5184} C_DIS
LIN {X -24.3551,Y -10.4402,Z 57,A -164.8792,B 24.8351,C -2.9619,E1 24.8517,E2 -472.2935} C_DIS
LIN {X -25.057,Y -8.6202,Z 57,A -169.1237,B 24.8338,C -2.9738,E1 24.8476,E2 -468.0535} C_DIS
LIN {X -25.6232,Y -6.7535,Z 57,A -173.3546,B 24.8324,C -2.9861,E1 24.8444,E2 -463.8276} C_DIS
LIN {X -26.0262,Y -4.9806,Z 57,A -177.3236,B 24.8311,C -2.9977,E1 24.8421,E2 -459.8629} C_DIS
LIN {X -26.3221,Y -3.0525,Z 57,A 178.4389,B 24.8297,C -3.0105,E1 24.8405,E2 -455.6308} C_DIS
LIN {X -26.4717,Y -1.1945,Z 57,A 174.3911,B 24.8282,C -3.0229,E1 24.8398,E2 -451.5883} C_DIS
LIN {X -26.4663,Y 1.3002,Z 57,A 168.9249,B 24.8264,C -3.0393,E1 24.8401,E2 -446.1284} C_DIS
LIN {X -26.2994,Y 3.2437,Z 57,A 164.6987,B 24.8249,C -3.0524,E1 24.8414,E2 -441.9083} C_DIS
LIN {X -25.9976,Y 5.1296,Z 57,A 160.5889,B 24.8234,C -3.0653,E1 24.8434,E2 -437.8051} C_DIS
LIN {X -25.5737,Y 6.9395,Z 57,A 156.4676,B 24.822,C -3.0771,E1 24.8462,E2 -433.6879} C_DIS
LIN {X -24.9939,Y 8.802,Z 57,A 152.1846,B 24.8206,C -3.0895,E1 24.8499,E2 -429.4101} C_DIS
LIN {X -24.2565,Y 10.6679,Z 57,A 147.8423,B 24.8191,C -3.1022,E1 24.8546,E2 -425.0743} C_DIS
LIN {X -23.3827,Y 12.4676,Z 57,A 143.4727,B 24.8176,C -3.1144,E1 24.8601,E2 -420.7103} C_DIS
LIN {X -22.4534,Y 14.072,Z 57,A 139.4236,B 24.8164,C -3.1252,E1 24.866,E2 -416.6664} C_DIS
LIN {X -21.3049,Y 15.7572,Z 57,A 134.9877,B 24.815,C -3.1368,E1 24.8731,E2 -412.2365} C_DIS
LIN {X -20.134,Y 17.2279,Z 57,A 130.882,B 24.8138,C -3.1468,E1 24.8804,E2 -408.1357} C_DIS
LIN {X -18.7377,Y 18.7377,Z 57,A 126.5451,B 24.8125,C -3.158,E1 24.8888,E2 -403.807} C_DIS
LIN {X -17.3577,Y 20.0223,Z 57,A 122.3163,B 24.8115,C -3.1662,E1 24.8975,E2 -399.5807} C_DIS
LIN {X -15.8878,Y 21.2074,Z 57,A 118.2245,B 24.8105,C -3.1745,E1 24.9066,E2 -395.4939} C_DIS
LIN {X -14.2217,Y 22.3591,Z 57,A 113.824,B 24.8095,C -3.1826,E1 24.9168,E2 -391.0983} C_DIS
LIN {X -12.4915,Y 23.3699,Z 57,A 109.4838,B 24.8086,C -3.1899,E1 24.9273,E2 -386.7629} C_DIS
LIN {X -10.7382,Y 24.225,Z 57,A 105.2656,B 24.8079,C -3.1962,E1 24.938,E2 -382.5492} C_DIS
LIN {X -8.927,Y 24.9493,Z 57,A 101.0437,B 24.8072,C -3.2016,E1 24.949,E2 -378.3313} C_DIS
LIN {X -7.0675,Y 25.5385,Z 57,A 96.8175,B 24.8067,C -3.206,E1 24.9603,E2 -374.1086} C_DIS
LIN {X -5.1696,Y 25.9896,Z 57,A 92.6086,B 24.8062,C -3.2097,E1 24.9718,E2 -369.9033} C_DIS
LIN {X -3.2909,Y 26.2937,Z 57,A 88.3782,B 24.806,C -3.2114,E1 24.9835,E2 -365.6735} C_DIS
LIN {X -1.3002,Y 26.4663,Z 57,A 84.1621,B 24.8057,C -3.214,E1 24.9952,E2 -361.462} C_DIS
LIN {X 0.6503,Y 26.4906,Z 57,A 79.8929,B 24.8057,C -3.2143,E1 25.0071,E2 -357.1939} C_DIS
LIN {X 2.5973,Y 26.3708,Z 57,A 75.716,B 24.8057,C -3.2144,E1 25.0187,E2 -353.0194} C_DIS
LIN {X 4.5145,Y 26.1116,Z 57,A 71.5423,B 24.8058,C -3.2133,E1 25.0303,E2 -348.847} C_DIS
LIN {X 6.3641,Y 25.7231,Z 57,A 67.4466,B 24.8061,C -3.2112,E1 25.0414,E2 -344.7519} C_DIS
LIN {X 8.2177,Y 25.1922,Z 57,A 63.2815,B 24.8064,C -3.2082,E1 25.0525,E2 -340.5871} C_DIS
LIN {X 10.046,Y 24.5205,Z 57,A 59.051,B 24.8069,C -3.204,E1 25.0635,E2 -336.356} C_DIS
LIN {X 11.7953,Y 23.7284,Z 57,A 54.9333,B 24.8075,C -3.1996,E1 25.0739,E2 -332.2384} C_DIS
LIN {X 13.509,Y 22.7965,Z 57,A 50.6982,B 24.8082,C -3.1936,E1 25.0842,E2 -328.0017} C_DIS
LIN {X 15.204,Y 21.703,Z 57,A 46.3346,B 24.809,C -3.1867,E1 25.0943,E2 -323.6364} C_DIS
LIN {X 16.8106,Y 20.4838,Z 57,A 42.1234,B 24.8098,C -3.1806,E1 25.1036,E2 -319.4262} C_DIS
LIN {X 18.1755,Y 19.2828,Z 57,A 38.1138,B 24.8108,C -3.1721,E1 25.1119,E2 -315.4127} C_DIS
LIN {X 19.5615,Y 17.8753,Z 57,A 33.8174,B 24.8119,C -3.1627,E1 25.1201,E2 -311.1127} C_DIS
LIN {X 20.8873,Y 16.307,Z 57,A 29.5318,B 24.8129,C -3.1543,E1 25.1277,E2 -306.8269} C_DIS
LIN {X 21.9917,Y 14.7834,Z 57,A 25.371,B 24.8142,C -3.1433,E1 25.1343,E2 -302.6605} C_DIS
LIN {X 23.0564,Y 13.0613,Z 57,A 21.0359,B 24.8155,C -3.1325,E1 25.1405,E2 -298.322} C_DIS
LIN {X 23.9543,Y 11.3295,Z 57,A 16.8527,B 24.8168,C -3.1215,E1 25.1457,E2 -294.1352} C_DIS
LIN {X 24.7227,Y 9.5366,Z 57,A 12.662,B 24.8182,C -3.11,E1 25.1501,E2 -289.9402} C_DIS
LIN {X 25.3572,Y 7.692,Z 57,A 8.477,B 24.8195,C -3.0981,E1 25.1537,E2 -285.7508} C_DIS
LIN {X 25.8547,Y 5.8059,Z 57,A 4.4171,B 24.8208,C -3.0874,E1 25.1564,E2 -281.689} C_DIS
LIN {X 26.192,Y 4.0193,Z 57,A 0.3739,B 24.8223,C -3.0742,E1 25.1583,E2 -277.6381} C_DIS
LIN {X 26.4158,Y 2.0929,Z 57,A -3.7025,B 24.8237,C -3.0626,E1 25.1595,E2 -273.5585} C_DIS
LIN {X 26.504,Y 0.0086,Z 57,A -8.3878,B 24.8255,C -3.0464,E1 25.1597,E2 -268.8628} C_DIS
LIN {X 26.4264,Y -1.9493,Z 57,A -12.4579,B 24.8268,C -3.0352,E1 25.1591,E2 -264.7903} C_DIS
LIN {X 26.1769,Y -4.1171,Z 57,A -16.1403,B 24.8271,C -3.0328,E1 25.1578,E2 -261.124} C_DIS
LIN {X 25.9976,Y -5.1296,Z 57,A -19.291,B 24.8292,C -3.0149,E1 25.1562,E2 -257.9492} C_DIS
LIN {X 25.5795,Y -6.9177,Z 57,A -23.3239,B 24.8306,C -3.0019,E1 25.1535,E2 -253.909} C_DIS
LIN {X 24.9939,Y -8.802,Z 57,A -27.5451,B 24.832,C -2.9896,E1 25.1498,E2 -249.6823} C_DIS
LIN {X 24.2565,Y -10.6679,Z 57,A -31.8594,B 24.8334,C -2.977,E1 25.1451,E2 -245.3619} C_DIS
LIN {X 23.3827,Y -12.4676,Z 57,A -36.1708,B 24.8348,C -2.9647,E1 25.1397,E2 -241.0443} C_DIS
LIN {X 22.4534,Y -14.072,Z 57,A -40.1678,B 24.8361,C -2.9537,E1 25.1339,E2 -237.0416} C_DIS
LIN {X 21.3049,Y -15.7572,Z 57,A -44.5489,B 24.8373,C -2.9422,E1 25.1268,E2 -232.6547} C_DIS
LIN {X 20.1456,Y -17.2143,Z 57,A -48.5635,B 24.8384,C -2.9321,E1 25.1196,E2 -228.6345} C_DIS
LIN {X 18.7377,Y -18.7377,Z 57,A -52.895,B 24.8395,C -2.923,E1 25.1113,E2 -224.3002} C_DIS
LIN {X 17.3577,Y -20.0223,Z 57,A -57.0798,B 24.8406,C -2.9126,E1 25.1026,E2 -220.1076} C_DIS
LIN {X 15.8878,Y -21.2074,Z 57,A -61.1322,B 24.8415,C -2.9044,E1 25.0936,E2 -216.0507} C_DIS
LIN {X 14.2217,Y -22.3591,Z 57,A -65.4939,B 24.8424,C -2.8962,E1 25.0835,E2 -211.6841} C_DIS
LIN {X 12.4915,Y -23.3699,Z 57,A -69.7945,B 24.8432,C -2.8891,E1 25.073,E2 -207.3793} C_DIS
LIN {X 10.7382,Y -24.225,Z 57,A -73.9883,B 24.8438,C -2.8829,E1 25.0624,E2 -203.1815} C_DIS
LIN {X 8.927,Y -24.9493,Z 57,A -78.1847,B 24.8444,C -2.8776,E1 25.0514,E2 -198.9815} C_DIS
LIN {X 7.0675,Y -25.5385,Z 57,A -82.3895,B 24.8449,C -2.873,E1 25.0401,E2 -194.7732} C_DIS
LIN {X 5.1696,Y -25.9896,Z 57,A -86.5813,B 24.8453,C -2.8695,E1 25.0287,E2 -190.5786} C_DIS
LIN {X 3.2909,Y -26.2937,Z 57,A -90.7989,B 24.8457,C -2.8658,E1 25.017,E2 -186.3559} C_DIS
LIN {X 1.3002,Y -26.4663,Z 57,A -95.0067,B 24.8457,C -2.865,E1 25.0053,E2 -182.1479} C_DIS
LIN {X 0.0182,Y -26.4948,Z 57,A -97.1641,B 24.8453,C -2.8698,E1 24.9993,E2 -180.0023} C_DIS
Enddeposition()
LIN {X 0.0182,Y -26.4948,Z 57,A -97.1641,B 24.8453,C -2.8698,E1 24.9993,E2 -180.0023} C_DIS
Startdeposition()
$VEL.CP = VEL_PRINT
LIN {X 1.0723,Y -25.4876,Z 57,A -93.4173,B 24.842,C -2.9,E1 25.01,E2 -183.8201} C_DIS
LIN {X 2.9462,Y -25.3395,Z 57,A -89.1613,B 24.8417,C -2.9025,E1 25.0218,E2 -188.0795} C_DIS
LIN {X 4.8092,Y -25.0528,Z 57,A -85.0261,B 24.8415,C -2.9048,E1 25.0332,E2 -192.2157} C_DIS
LIN {X 6.5945,Y -24.6429,Z 57,A -81.4707,B 24.8416,C -2.9034,E1 25.0428,E2 -195.7627} C_DIS
LIN {X 8.0821,Y -24.1958,Z 57,A -77.2413,B 24.8404,C -2.9147,E1 25.0541,E2 -200.011} C_DIS
LIN {X 9.5903,Y -23.6387,Z 57,A -73.9912,B 24.8402,C -2.9159,E1 25.0625,E2 -203.257} C_DIS
LIN {X 11.3355,Y -22.8533,Z 57,A -69.4783,B 24.8393,C -2.9247,E1 25.074,E2 -207.7791} C_DIS
LIN {X 12.7075,Y -22.12,Z 57,A -65.9912,B 24.8386,C -2.9306,E1 25.0825,E2 -211.27} C_DIS
LIN {X 14.345,Y -21.095,Z 57,A -62.3949,B 24.8386,C -2.931,E1 25.0909,E2 -214.8554} C_DIS
LIN {X 15.8135,Y -20.0178,Z 57,A -57.0613,B 24.8361,C -2.9528,E1 25.1028,E2 -220.2213} C_DIS
LIN {X 17.5268,Y -18.5361,Z 57,A -52.0043,B 24.8349,C -2.964,E1 25.1132,E2 -225.2845} C_DIS
LIN {X 19.6833,Y -16.2282,Z 57,A -45.4108,B 24.8336,C -2.9759,E1 25.1255,E2 -231.8768} C_DIS
LIN {X 20.7825,Y -14.7941,Z 57,A -41.2226,B 24.8322,C -2.9881,E1 25.1324,E2 -236.0738} C_DIS
LIN {X 21.9517,Y -12.9962,Z 57,A -36.6777,B 24.831,C -2.9984,E1 25.1391,E2 -240.6198} C_DIS
LIN {X 22.8592,Y -11.3234,Z 57,A -32.4192,B 24.8297,C -3.0104,E1 25.1446,E2 -244.8844} C_DIS
Enddeposition()
END
